LIN {X 0,Y 312.688,Z 247.371,A -85,B 0,C 180,E1 -15958.713,E2 -15958.713} C_VEL
LIN {X 0,Y 312.385,Z 243.779,A -85,B 0,C 180,E1 -15959.666,E2 -15959.666} C_VEL
LIN {X 0,Y 310.267,Z 233.599,A -85,B 0,C 180,E1 -15962.611,E2 -15962.611} C_VEL
LIN {X 0,Y 307.607,Z 223.567,A -85,B 0,C 180,E1 -15965.799,E2 -15965.799} C_VEL
LIN {X 0,Y 305.424,Z 216.441,A -85,B 0,C 180,E1 -15968.279,E2 -15968.279} C_VEL
LIN {X 0,Y 305.436,Z 216.435,A -85,B 0,C 180,E1 -15972.581,E2 -15972.581} C_VEL
LIN {X 0,Y 305.421,Z 216.44,A -85,B 0,C 180,E1 -15976.344,E2 -15976.344} C_VEL
LIN {X 0,Y 305.409,Z 216.437,A -85,B 0,C 180,E1 -15979.884,E2 -15979.884} C_VEL
LIN {X 0,Y 305.462,Z 216.436,A -85,B 0,C 180,E1 -15983.636,E2 -15983.636} C_VEL
LIN {X 0,Y 305.464,Z 216.436,A -85,B 0,C 180,E1 -15986.483,E2 -15986.483} C_VEL
LIN {X 0,Y 305.433,Z 216.439,A -85,B 0,C 180,E1 -15989.587,E2 -15989.587} C_VEL
LIN {X 0,Y 305.466,Z 216.432,A -85,B 0,C 180,E1 -15992.603,E2 -15992.603} C_VEL
LIN {X 0,Y 305.486,Z 216.432,A -85,B 0,C 180,E1 -15995.537,E2 -15995.537} C_VEL
LIN {X 0,Y 305.5,Z 216.426,A -85,B 0,C 180,E1 -15999.814,E2 -15999.814} C_VEL
LIN {X 0,Y 305.546,Z 216.418,A -85,B 0,C 180,E1 -16002.601,E2 -16002.601} C_VEL
LIN {X 0,Y 305.626,Z 216.409,A -85,B 0,C 180,E1 -16005.348,E2 -16005.348} C_VEL
LIN {X 0,Y 305.635,Z 216.412,A -85,B 0,C 180,E1 -16009.4,E2 -16009.4} C_VEL
LIN {X 0,Y 305.797,Z 216.394,A -85,B 0,C 180,E1 -16012.074,E2 -16012.074} C_VEL
LIN {X 0,Y 305.685,Z 216.407,A -85,B 0,C 180,E1 -16014.723,E2 -16014.723} C_VEL
LIN {X 0,Y 305.955,Z 216.371,A -85,B 0,C 180,E1 -16018.684,E2 -16018.684} C_VEL
LIN {X 0,Y 305.955,Z 216.375,A -85,B 0,C 180,E1 -16021.316,E2 -16021.316} C_VEL
LIN {X 0,Y 305.676,Z 216.41,A -85,B 0,C 180,E1 -16025.277,E2 -16025.277} C_VEL
LIN {X 0,Y 305.768,Z 216.397,A -85,B 0,C 180,E1 -16027.927,E2 -16027.927} C_VEL
LIN {X 0,Y 305.773,Z 216.514,A -85,B 0,C 180,E1 -16028.46,E2 -16028.46} C_VEL
LIN {X 0,Y 306.843,Z 219.417,A -85,B 0,C 180,E1 -16028.732,E2 -16028.732} C_VEL
LIN {X 0,Y 308.362,Z 221.654,A -85,B 0,C 180,E1 -16029.043,E2 -16029.043} C_VEL
LIN {X 0,Y 315.915,Z 234.684,A -85,B 0,C 180,E1 -16030.554,E2 -16030.554} C_VEL
LIN {X 0,Y 322.045,Z 246.925,A -85,B 0,C 180,E1 -16031.739,E2 -16031.739} C_VEL
LIN {X 0,Y 323.047,Z 249.102,A -85,B 0,C 180,E1 -16031.928,E2 -16031.928} C_VEL
LIN {X 0,Y 319.984,Z 321.185,A -85,B 0,C 180,E1 -16033.904,E2 -16033.904} C_VEL
LIN {X 0,Y 319.265,Z 334.155,A -85,B 0,C 180,E1 -16034.524,E2 -16034.524} C_VEL
LIN {X 0,Y 318.134,Z 346.76,A -85,B 0,C 180,E1 -16035.373,E2 -16035.373} C_VEL
LIN {X 0,Y 316.667,Z 358.574,A -85,B 0,C 180,E1 -16036.437,E2 -16036.437} C_VEL
LIN {X 0,Y 315.006,Z 370.51,A -85,B 0,C 180,E1 -16037.832,E2 -16037.832} C_VEL
LIN {X 0,Y 313.265,Z 380.5,A -85,B 0,C 180,E1 -16039.301,E2 -16039.301} C_VEL
LIN {X 0,Y 311.413,Z 390.569,A -85,B 0,C 180,E1 -16041.167,E2 -16041.167} C_VEL
LIN {X 0,Y 309.756,Z 398.606,A -85,B 0,C 180,E1 -16043.04,E2 -16043.04} C_VEL
LIN {X 0,Y 308.28,Z 405.247,A -85,B 0,C 180,E1 -16044.985,E2 -16044.985} C_VEL
LIN {X 0,Y 306.948,Z 411.266,A -85,B 0,C 180,E1 -16047.253,E2 -16047.253} C_VEL
LIN {X 0,Y 305.986,Z 415.201,A -85,B 0,C 180,E1 -16049.215,E2 -16049.215} C_VEL
LIN {X 0,Y 305.093,Z 418.533,A -85,B 0,C 180,E1 -16051.536,E2 -16051.536} C_VEL
LIN {X 0,Y 304.455,Z 420.465,A -85,B 0,C 180,E1 -16053.797,E2 -16053.797} C_VEL
LIN {X 0,Y 304.084,Z 421.192,A -85,B 0,C 180,E1 -16056.01,E2 -16056.01} C_VEL
LIN {X 0,Y 303.898,Z 420.598,A -85,B 0,C 180,E1 -16058.639,E2 -16058.639} C_VEL
LIN {X 0,Y 303.963,Z 419.321,A -85,B 0,C 180,E1 -16060.346,E2 -16060.346} C_VEL
LIN {X 0,Y 304.211,Z 416.972,A -85,B 0,C 180,E1 -16062.331,E2 -16062.331} C_VEL
LIN {X 0,Y 304.581,Z 413.591,A -85,B 0,C 180,E1 -16064.332,E2 -16064.332} C_VEL
LIN {X 0,Y 305.07,Z 409.227,A -85,B 0,C 180,E1 -16066.282,E2 -16066.282} C_VEL
LIN {X 0,Y 305.647,Z 403.845,A -85,B 0,C 180,E1 -16068.178,E2 -16068.178} C_VEL
LIN {X 0,Y 306.511,Z 396.159,A -85,B 0,C 180,E1 -16070.333,E2 -16070.333} C_VEL
LIN {X 0,Y 307.543,Z 387.805,A -85,B 0,C 180,E1 -16072.185,E2 -16072.185} C_VEL
LIN {X 0,Y 308.695,Z 377.652,A -85,B 0,C 180,E1 -16074.002,E2 -16074.002} C_VEL
LIN {X 0,Y 309.71,Z 367.705,A -85,B 0,C 180,E1 -16075.438,E2 -16075.438} C_VEL
LIN {X 0,Y 310.869,Z 356.07,A -85,B 0,C 180,E1 -16076.77,E2 -16076.77} C_VEL
LIN {X 0,Y 311.902,Z 343.287,A -85,B 0,C 180,E1 -16077.911,E2 -16077.911} C_VEL
LIN {X 0,Y 312.629,Z 329.893,A -85,B 0,C 180,E1 -16078.784,E2 -16078.784} C_VEL
LIN {X 0,Y 313.199,Z 316.6,A -85,B 0,C 180,E1 -16079.374,E2 -16079.374} C_VEL
LIN {X 0,Y 315.113,Z 241.687,A -85,B 0,C 180,E1 -16081.346,E2 -16081.346} C_VEL
LIN {X 0,Y 305.539,Z 216.426,A -85,B 0,C 180,E1 -16082.7,E2 -16082.7} C_VEL
LIN {X 0,Y 305.505,Z 216.429,A -85,B 0,C 180,E1 -16085.539,E2 -16085.539} C_VEL
LIN {X 0,Y 305.497,Z 216.429,A -85,B 0,C 180,E1 -16089.814,E2 -16089.814} C_VEL
LIN {X 0,Y 305.545,Z 216.425,A -85,B 0,C 180,E1 -16092.602,E2 -16092.602} C_VEL
LIN {X 0,Y 305.627,Z 216.414,A -85,B 0,C 180,E1 -16095.348,E2 -16095.348} C_VEL
LIN {X 0,Y 305.625,Z 216.413,A -85,B 0,C 180,E1 -16099.4,E2 -16099.4} C_VEL
LIN {X 0,Y 305.75,Z 216.398,A -85,B 0,C 180,E1 -16102.073,E2 -16102.073} C_VEL
LIN {X 0,Y 305.672,Z 216.411,A -85,B 0,C 180,E1 -16104.724,E2 -16104.724} C_VEL
LIN {X 0,Y 305.953,Z 216.375,A -85,B 0,C 180,E1 -16108.684,E2 -16108.684} C_VEL
LIN {X 0,Y 305.953,Z 216.371,A -85,B 0,C 180,E1 -16111.317,E2 -16111.317} C_VEL
LIN {X 0,Y 305.669,Z 216.407,A -85,B 0,C 180,E1 -16115.277,E2 -16115.277} C_VEL
LIN {X 0,Y 305.765,Z 216.397,A -85,B 0,C 180,E1 -16117.927,E2 -16117.927} C_VEL
LIN {X 0,Y 305.605,Z 216.417,A -85,B 0,C 180,E1 -16121.945,E2 -16121.945} C_VEL
LIN {X 0,Y 305.64,Z 216.41,A -85,B 0,C 180,E1 -16125.035,E2 -16125.035} C_VEL
LIN {X 0,Y 305.581,Z 216.417,A -85,B 0,C 180,E1 -16128.783,E2 -16128.783} C_VEL
LIN {X 0,Y 305.488,Z 216.428,A -85,B 0,C 180,E1 -16133.04,E2 -16133.04} C_VEL
LIN {X 0,Y 305.477,Z 216.433,A -85,B 0,C 180,E1 -16136.2,E2 -16136.2} C_VEL
LIN {X 0,Y 305.46,Z 216.433,A -85,B 0,C 180,E1 -16139.038,E2 -16139.038} C_VEL
LIN {X 0,Y 305.438,Z 216.438,A -85,B 0,C 180,E1 -16141.953,E2 -16141.953} C_VEL
LIN {X 0,Y 305.464,Z 216.432,A -85,B 0,C 180,E1 -16145.114,E2 -16145.114} C_VEL
LIN {X 0,Y 305.428,Z 216.433,A -85,B 0,C 180,E1 -16148.524,E2 -16148.524} C_VEL
LIN {X 0,Y 305.429,Z 216.438,A -85,B 0,C 180,E1 -16151.859,E2 -16151.859} C_VEL
LIN {X 0,Y 305.401,Z 216.445,A -85,B 0,C 180,E1 -16155.511,E2 -16155.511} C_VEL
LIN {X 0,Y 305.414,Z 216.439,A -85,B 0,C 180,E1 -16158.139,E2 -16158.139} C_VEL
LIN {X 0,Y 305.462,Z 216.434,A -85,B 0,C 180,E1 -16161.595,E2 -16161.595} C_VEL
LIN {X 0,Y 305.464,Z 216.434,A -85,B 0,C 180,E1 -16164.887,E2 -16164.887} C_VEL
LIN {X 0,Y 305.434,Z 216.433,A -85,B 0,C 180,E1 -16166.96,E2 -16166.96} C_VEL
LIN {X 0,Y 304.738,Z 216.524,A -85,B 0,C 180,E1 -16168.061,E2 -16168.061} C_VEL
LIN {X 0,Y 301.878,Z 216.879,A -85,B 0,C 180,E1 -16169.854,E2 -16169.854} C_VEL
LIN {X 0,Y 299.48,Z 217.18,A -85,B 0,C 180,E1 -16171.309,E2 -16171.309} C_VEL
LIN {X 0,Y 298.464,Z 217.305,A -85,B 0,C 180,E1 -16172.435,E2 -16172.435} C_VEL
LIN {X 0,Y 298.387,Z 217.311,A -85,B 0,C 180,E1 -16172.816,E2 -16172.816} C_VEL
LIN {X 0,Y 298.423,Z 217.309,A -85,B 0,C 180,E1 -16176.399,E2 -16176.399} C_VEL
LIN {X 0,Y 298.509,Z 217.303,A -85,B 0,C 180,E1 -16180.755,E2 -16180.755} C_VEL
LIN {X 0,Y 298.589,Z 217.29,A -85,B 0,C 180,E1 -16184.995,E2 -16184.995} C_VEL
LIN {X 0,Y 298.586,Z 217.285,A -85,B 0,C 180,E1 -16189.146,E2 -16189.146} C_VEL
LIN {X 0,Y 298.701,Z 217.271,A -85,B 0,C 180,E1 -16191.884,E2 -16191.884} C_VEL
LIN {X 0,Y 298.637,Z 217.286,A -85,B 0,C 180,E1 -16194.599,E2 -16194.599} C_VEL
LIN {X 0,Y 298.91,Z 217.252,A -85,B 0,C 180,E1 -16198.653,E2 -16198.653} C_VEL
LIN {X 0,Y 298.915,Z 217.248,A -85,B 0,C 180,E1 -16201.347,E2 -16201.347} C_VEL
LIN {X 0,Y 298.738,Z 217.268,A -85,B 0,C 180,E1 -16206.755,E2 -16206.755} C_VEL
LIN {X 0,Y 298.633,Z 217.281,A -85,B 0,C 180,E1 -16209.482,E2 -16209.482} C_VEL
LIN {X 0,Y 298.527,Z 217.298,A -85,B 0,C 180,E1 -16213.617,E2 -16213.617} C_VEL
LIN {X 0,Y 298.5,Z 217.304,A -85,B 0,C 180,E1 -16217.823,E2 -16217.823} C_VEL
LIN {X 0,Y 298.428,Z 217.307,A -85,B 0,C 180,E1 -16220.686,E2 -16220.686} C_VEL
LIN {X 0,Y 298.424,Z 217.31,A -85,B 0,C 180,E1 -16225.082,E2 -16225.082} C_VEL
LIN {X 0,Y 298.404,Z 217.314,A -85,B 0,C 180,E1 -16229.375,E2 -16229.375} C_VEL
LIN {X 0,Y 298.395,Z 217.313,A -85,B 0,C 180,E1 -16232.8,E2 -16232.8} C_VEL
LIN {X 0,Y 298.43,Z 217.309,A -85,B 0,C 180,E1 -16236.803,E2 -16236.803} C_VEL
LIN {X 0,Y 298.376,Z 217.321,A -85,B 0,C 180,E1 -16239.492,E2 -16239.492} C_VEL
LIN {X 0,Y 298.372,Z 217.319,A -85,B 0,C 180,E1 -16243.097,E2 -16243.097} C_VEL
LIN {X 0,Y 298.373,Z 217.318,A -85,B 0,C 180,E1 -16246.915,E2 -16246.915} C_VEL
LIN {X 0,Y 298.387,Z 217.318,A -85,B 0,C 180,E1 -16251.011,E2 -16251.011} C_VEL
LIN {X 0,Y 298.409,Z 217.312,A -85,B 0,C 180,E1 -16253.928,E2 -16253.928} C_VEL
LIN {X 0,Y 298.47,Z 217.477,A -85,B 0,C 180,E1 -16255.589,E2 -16255.589} C_VEL
LIN {X 0,Y 301.208,Z 230.094,A -85,B 0,C 180,E1 -16259.114,E2 -16259.114} C_VEL
LIN {X 0,Y 303.252,Z 240.673,A -85,B 0,C 180,E1 -16261.947,E2 -16261.947} C_VEL
LIN {X 0,Y 301.833,Z 252.558,A -85,B 0,C 180,E1 -16264.843,E2 -16264.843} C_VEL
LIN {X 0,Y 307.37,Z 301.3,A -85,B 0,C 180,E1 -16266.603,E2 -16266.603} C_VEL
LIN {X 0,Y 305.725,Z 362.778,A -85,B 0,C 180,E1 -16268.286,E2 -16268.286} C_VEL
LIN {X 0,Y 304.805,Z 376.523,A -85,B 0,C 180,E1 -16268.927,E2 -16268.927} C_VEL
LIN {X 0,Y 303.869,Z 387.983,A -85,B 0,C 180,E1 -16269.7,E2 -16269.7} C_VEL
LIN {X 0,Y 302.703,Z 399.031,A -85,B 0,C 180,E1 -16270.679,E2 -16270.679} C_VEL
LIN {X 0,Y 301.341,Z 410.628,A -85,B 0,C 180,E1 -16271.999,E2 -16271.999} C_VEL
LIN {X 0,Y 300.091,Z 421.14,A -85,B 0,C 180,E1 -16273.503,E2 -16273.503} C_VEL
LIN {X 0,Y 299.107,Z 429.755,A -85,B 0,C 180,E1 -16275.021,E2 -16275.021} C_VEL
LIN {X 0,Y 298.111,Z 439.072,A -85,B 0,C 180,E1 -16277.058,E2 -16277.058} C_VEL
LIN {X 0,Y 297.307,Z 446.538,A -85,B 0,C 180,E1 -16279.099,E2 -16279.099} C_VEL
LIN {X 0,Y 296.966,Z 452.512,A -85,B 0,C 180,E1 -16281.151,E2 -16281.151} C_VEL
LIN {X 0,Y 296.848,Z 457.164,A -85,B 0,C 180,E1 -16283.201,E2 -16283.201} C_VEL
LIN {X 0,Y 296.877,Z 459.588,A -85,B 0,C 180,E1 -16284.566,E2 -16284.566} C_VEL
LIN {X 0,Y 296.844,Z 461.54,A -85,B 0,C 180,E1 -16285.927,E2 -16285.927} C_VEL
LIN {X 0,Y 296.928,Z 463.054,A -85,B 0,C 180,E1 -16287.286,E2 -16287.286} C_VEL
LIN {X 0,Y 297.085,Z 464.085,A -85,B 0,C 180,E1 -16288.644,E2 -16288.644} C_VEL
LIN {X 0,Y 297.089,Z 464.68,A -85,B 0,C 180,E1 -16290,E2 -16290} C_VEL
LIN {X 0,Y 297.049,Z 464.857,A -85,B 0,C 180,E1 -16291.355,E2 -16291.355} C_VEL
LIN {X 0,Y 296.81,Z 464.596,A -85,B 0,C 180,E1 -16292.714,E2 -16292.714} C_VEL
LIN {X 0,Y 296.759,Z 463.895,A -85,B 0,C 180,E1 -16294.074,E2 -16294.074} C_VEL
LIN {X 0,Y 296.649,Z 462.52,A -85,B 0,C 180,E1 -16295.71,E2 -16295.71} C_VEL
LIN {X 0,Y 296.84,Z 459.301,A -85,B 0,C 180,E1 -16298.167,E2 -16298.167} C_VEL
LIN {X 0,Y 297.197,Z 455.495,A -85,B 0,C 180,E1 -16300.215,E2 -16300.215} C_VEL
LIN {X 0,Y 297.889,Z 450.586,A -85,B 0,C 180,E1 -16302.259,E2 -16302.259} C_VEL
LIN {X 0,Y 299.293,Z 443.267,A -85,B 0,C 180,E1 -16304.621,E2 -16304.621} C_VEL
LIN {X 0,Y 300.685,Z 435.56,A -85,B 0,C 180,E1 -16306.602,E2 -16306.602} C_VEL
LIN {X 0,Y 302.319,Z 427.464,A -85,B 0,C 180,E1 -16308.29,E2 -16308.29} C_VEL
LIN {X 0,Y 304.475,Z 416.739,A -85,B 0,C 180,E1 -16310.081,E2 -16310.081} C_VEL
LIN {X 0,Y 306.557,Z 405.968,A -85,B 0,C 180,E1 -16311.519,E2 -16311.519} C_VEL
LIN {X 0,Y 308.314,Z 395.683,A -85,B 0,C 180,E1 -16312.623,E2 -16312.623} C_VEL
LIN {X 0,Y 310.192,Z 383.601,A -85,B 0,C 180,E1 -16313.624,E2 -16313.624} C_VEL
LIN {X 0,Y 311.711,Z 371.311,A -85,B 0,C 180,E1 -16314.386,E2 -16314.386} C_VEL
LIN {X 0,Y 312.826,Z 358.25,A -85,B 0,C 180,E1 -16314.957,E2 -16314.957} C_VEL
LIN {X 0,Y 315.076,Z 301.694,A -85,B 0,C 180,E1 -16316.543,E2 -16316.543} C_VEL
LIN {X 0,Y 312.642,Z 279.918,A -85,B 0,C 180,E1 -16317.569,E2 -16317.569} C_VEL
LIN {X 0,Y 309.361,Z 260.607,A -85,B 0,C 180,E1 -16318.667,E2 -16318.667} C_VEL
LIN {X 0,Y 306.799,Z 249.329,A -85,B 0,C 180,E1 -16319.425,E2 -16319.425} C_VEL
LIN {X 0,Y 305.838,Z 246.569,A -85,B 0,C 180,E1 -16319.712,E2 -16319.712} C_VEL
LIN {X 0,Y 303.74,Z 236.256,A -85,B 0,C 180,E1 -16322.775,E2 -16322.775} C_VEL
LIN {X 0,Y 301.472,Z 227.417,A -85,B 0,C 180,E1 -16325.648,E2 -16325.648} C_VEL
LIN {X 0,Y 298.972,Z 219.432,A -85,B 0,C 180,E1 -16328.521,E2 -16328.521} C_VEL
LIN {X 0,Y 298.356,Z 217.318,A -85,B 0,C 180,E1 -16329.337,E2 -16329.337} C_VEL
LIN {X 0,Y 298.371,Z 217.314,A -85,B 0,C 180,E1 -16333.097,E2 -16333.097} C_VEL
LIN {X 0,Y 298.371,Z 217.314,A -85,B 0,C 180,E1 -16336.915,E2 -16336.915} C_VEL
LIN {X 0,Y 298.384,Z 217.318,A -85,B 0,C 180,E1 -16341.011,E2 -16341.011} C_VEL
LIN {X 0,Y 298.405,Z 217.316,A -85,B 0,C 180,E1 -16343.928,E2 -16343.928} C_VEL
LIN {X 0,Y 298.392,Z 217.312,A -85,B 0,C 180,E1 -16347.199,E2 -16347.199} C_VEL
LIN {X 0,Y 298.407,Z 217.308,A -85,B 0,C 180,E1 -16350.623,E2 -16350.623} C_VEL
LIN {X 0,Y 298.447,Z 217.309,A -85,B 0,C 180,E1 -16354.92,E2 -16354.92} C_VEL
LIN {X 0,Y 298.432,Z 217.306,A -85,B 0,C 180,E1 -16359.314,E2 -16359.314} C_VEL
LIN {X 0,Y 298.507,Z 217.296,A -85,B 0,C 180,E1 -16362.177,E2 -16362.177} C_VEL
LIN {X 0,Y 298.585,Z 217.287,A -85,B 0,C 180,E1 -16364.994,E2 -16364.994} C_VEL
LIN {X 0,Y 298.591,Z 217.288,A -85,B 0,C 180,E1 -16369.146,E2 -16369.146} C_VEL
LIN {X 0,Y 298.741,Z 217.271,A -85,B 0,C 180,E1 -16371.885,E2 -16371.885} C_VEL
LIN {X 0,Y 298.656,Z 217.283,A -85,B 0,C 180,E1 -16374.599,E2 -16374.599} C_VEL
LIN {X 0,Y 298.922,Z 217.247,A -85,B 0,C 180,E1 -16378.653,E2 -16378.653} C_VEL
LIN {X 0,Y 298.922,Z 217.251,A -85,B 0,C 180,E1 -16381.347,E2 -16381.347} C_VEL
LIN {X 0,Y 298.72,Z 217.274,A -85,B 0,C 180,E1 -16386.515,E2 -16386.515} C_VEL
LIN {X 0,Y 298.735,Z 217.275,A -85,B 0,C 180,E1 -16387.349,E2 -16387.349} C_VEL
LIN {X 0,Y 299.806,Z 220.259,A -85,B 0,C 180,E1 -16387.662,E2 -16387.662} C_VEL
LIN {X 0,Y 301.416,Z 222.354,A -85,B 0,C 180,E1 -16388,E2 -16388} C_VEL
LIN {X 0,Y 310.025,Z 237.229,A -85,B 0,C 180,E1 -16389.843,E2 -16389.843} C_VEL
LIN {X 0,Y 316.356,Z 249.735,A -85,B 0,C 180,E1 -16391.123,E2 -16391.123} C_VEL
LIN {X 0,Y 317.022,Z 251.251,A -85,B 0,C 180,E1 -16391.261,E2 -16391.261} C_VEL
LIN {X 0,Y 313.904,Z 322.243,A -85,B 0,C 180,E1 -16393.267,E2 -16393.267} C_VEL
LIN {X 0,Y 313.163,Z 334.721,A -85,B 0,C 180,E1 -16393.878,E2 -16393.878} C_VEL
LIN {X 0,Y 311.958,Z 347.565,A -85,B 0,C 180,E1 -16394.761,E2 -16394.761} C_VEL
LIN {X 0,Y 310.296,Z 360.242,A -85,B 0,C 180,E1 -16395.939,E2 -16395.939} C_VEL
LIN {X 0,Y 308.695,Z 370.876,A -85,B 0,C 180,E1 -16397.216,E2 -16397.216} C_VEL
LIN {X 0,Y 306.904,Z 380.791,A -85,B 0,C 180,E1 -16398.699,E2 -16398.699} C_VEL
LIN {X 0,Y 304.949,Z 390.754,A -85,B 0,C 180,E1 -16400.577,E2 -16400.577} C_VEL
LIN {X 0,Y 303.053,Z 399.391,A -85,B 0,C 180,E1 -16402.624,E2 -16402.624} C_VEL
LIN {X 0,Y 301.351,Z 406.616,A -85,B 0,C 180,E1 -16404.821,E2 -16404.821} C_VEL
LIN {X 0,Y 299.976,Z 412.353,A -85,B 0,C 180,E1 -16407.092,E2 -16407.092} C_VEL
LIN {X 0,Y 298.761,Z 416.929,A -85,B 0,C 180,E1 -16409.604,E2 -16409.604} C_VEL
LIN {X 0,Y 297.919,Z 419.716,A -85,B 0,C 180,E1 -16411.87,E2 -16411.87} C_VEL
LIN {X 0,Y 297.231,Z 421.484,A -85,B 0,C 180,E1 -16414.574,E2 -16414.574} C_VEL
LIN {X 0,Y 296.957,Z 421.761,A -85,B 0,C 180,E1 -16416.422,E2 -16416.422} C_VEL
LIN {X 0,Y 296.822,Z 421.096,A -85,B 0,C 180,E1 -16418.615,E2 -16418.615} C_VEL
LIN {X 0,Y 296.907,Z 419.404,A -85,B 0,C 180,E1 -16420.759,E2 -16420.759} C_VEL
LIN {X 0,Y 297.307,Z 416.024,A -85,B 0,C 180,E1 -16423.277,E2 -16423.277} C_VEL
LIN {X 0,Y 297.669,Z 412.624,A -85,B 0,C 180,E1 -16425.097,E2 -16425.097} C_VEL
LIN {X 0,Y 298.273,Z 406.939,A -85,B 0,C 180,E1 -16427.411,E2 -16427.411} C_VEL
LIN {X 0,Y 298.956,Z 401.062,A -85,B 0,C 180,E1 -16429.293,E2 -16429.293} C_VEL
LIN {X 0,Y 300.017,Z 392.542,A -85,B 0,C 180,E1 -16431.473,E2 -16431.473} C_VEL
LIN {X 0,Y 301.055,Z 383.725,A -85,B 0,C 180,E1 -16433.272,E2 -16433.272} C_VEL
LIN {X 0,Y 302.261,Z 373.726,A -85,B 0,C 180,E1 -16434.926,E2 -16434.926} C_VEL
LIN {X 0,Y 303.359,Z 362.693,A -85,B 0,C 180,E1 -16436.391,E2 -16436.391} C_VEL
LIN {X 0,Y 304.496,Z 350.668,A -85,B 0,C 180,E1 -16437.644,E2 -16437.644} C_VEL
LIN {X 0,Y 305.392,Z 338.484,A -85,B 0,C 180,E1 -16438.623,E2 -16438.623} C_VEL
LIN {X 0,Y 305.993,Z 324.851,A -85,B 0,C 180,E1 -16439.411,E2 -16439.411} C_VEL
LIN {X 0,Y 306.502,Z 311.68,A -85,B 0,C 180,E1 -16439.896,E2 -16439.896} C_VEL
LIN {X 0,Y 308.451,Z 243.989,A -85,B 0,C 180,E1 -16441.693,E2 -16441.693} C_VEL
LIN {X 0,Y 302.906,Z 228.819,A -85,B 0,C 180,E1 -16442.493,E2 -16442.493} C_VEL
LIN {X 0,Y 298.655,Z 218.077,A -85,B 0,C 180,E1 -16443.103,E2 -16443.103} C_VEL
LIN {X 0,Y 298.53,Z 217.3,A -85,B 0,C 180,E1 -16443.175,E2 -16443.175} C_VEL
LIN {X 0,Y 298.431,Z 217.312,A -85,B 0,C 180,E1 -16446.7,E2 -16446.7} C_VEL
LIN {X 0,Y 298.506,Z 217.303,A -85,B 0,C 180,E1 -16450.755,E2 -16450.755} C_VEL
LIN {X 0,Y 298.586,Z 217.293,A -85,B 0,C 180,E1 -16454.995,E2 -16454.995} C_VEL
LIN {X 0,Y 298.584,Z 217.292,A -85,B 0,C 180,E1 -16459.147,E2 -16459.147} C_VEL
LIN {X 0,Y 298.701,Z 217.275,A -85,B 0,C 180,E1 -16461.885,E2 -16461.885} C_VEL
LIN {X 0,Y 298.64,Z 217.287,A -85,B 0,C 180,E1 -16464.599,E2 -16464.599} C_VEL
LIN {X 0,Y 298.92,Z 217.252,A -85,B 0,C 180,E1 -16468.653,E2 -16468.653} C_VEL
LIN {X 0,Y 298.919,Z 217.247,A -85,B 0,C 180,E1 -16471.348,E2 -16471.348} C_VEL
LIN {X 0,Y 298.747,Z 217.271,A -85,B 0,C 180,E1 -16476.755,E2 -16476.755} C_VEL
LIN {X 0,Y 298.632,Z 217.283,A -85,B 0,C 180,E1 -16479.482,E2 -16479.482} C_VEL
LIN {X 0,Y 298.554,Z 217.294,A -85,B 0,C 180,E1 -16483.616,E2 -16483.616} C_VEL
LIN {X 0,Y 298.55,Z 217.296,A -85,B 0,C 180,E1 -16486.409,E2 -16486.409} C_VEL
LIN {X 0,Y 298.499,Z 217.301,A -85,B 0,C 180,E1 -16489.648,E2 -16489.648} C_VEL
LIN {X 0,Y 298.426,Z 217.309,A -85,B 0,C 180,E1 -16493.601,E2 -16493.601} C_VEL
LIN {X 0,Y 298.415,Z 217.311,A -85,B 0,C 180,E1 -16496.582,E2 -16496.582} C_VEL
LIN {X 0,Y 298.399,Z 217.316,A -85,B 0,C 180,E1 -16499.644,E2 -16499.644} C_VEL
LIN {X 0,Y 298.394,Z 217.312,A -85,B 0,C 180,E1 -16502.801,E2 -16502.801} C_VEL
LIN {X 0,Y 298.43,Z 217.305,A -85,B 0,C 180,E1 -16506.803,E2 -16506.803} C_VEL
LIN {X 0,Y 298.383,Z 217.313,A -85,B 0,C 180,E1 -16511.087,E2 -16511.087} C_VEL
LIN {X 0,Y 298.401,Z 217.313,A -85,B 0,C 180,E1 -16513.104,E2 -16513.104} C_VEL
LIN {X 0,Y 298.373,Z 217.317,A -85,B 0,C 180,E1 -16516.915,E2 -16516.915} C_VEL
LIN {X 0,Y 298.386,Z 217.316,A -85,B 0,C 180,E1 -16521.011,E2 -16521.011} C_VEL
LIN {X 0,Y 298.418,Z 217.309,A -85,B 0,C 180,E1 -16523.93,E2 -16523.93} C_VEL
LIN {X 0,Y 298.395,Z 217.318,A -85,B 0,C 180,E1 -16527.2,E2 -16527.2} C_VEL
LIN {X 0,Y 298.405,Z 217.313,A -85,B 0,C 180,E1 -16530.625,E2 -16530.625} C_VEL
LIN {X 0,Y 298.387,Z 217.311,A -85,B 0,C 180,E1 -16532.816,E2 -16532.816} C_VEL
LIN {X 0,Y 297.737,Z 217.396,A -85,B 0,C 180,E1 -16533.943,E2 -16533.943} C_VEL
LIN {X 0,Y 294.9,Z 217.759,A -85,B 0,C 180,E1 -16535.779,E2 -16535.779} C_VEL
LIN {X 0,Y 292.484,Z 218.062,A -85,B 0,C 180,E1 -16537.269,E2 -16537.269} C_VEL
LIN {X 0,Y 291.446,Z 218.186,A -85,B 0,C 180,E1 -16538.423,E2 -16538.423} C_VEL
LIN {X 0,Y 291.361,Z 218.193,A -85,B 0,C 180,E1 -16538.814,E2 -16538.814} C_VEL
LIN {X 0,Y 291.444,Z 218.178,A -85,B 0,C 180,E1 -16541.731,E2 -16541.731} C_VEL
LIN {X 0,Y 291.519,Z 218.168,A -85,B 0,C 180,E1 -16546.05,E2 -16546.05} C_VEL
LIN {X 0,Y 291.571,Z 218.159,A -85,B 0,C 180,E1 -16550.286,E2 -16550.286} C_VEL
LIN {X 0,Y 291.691,Z 218.146,A -85,B 0,C 180,E1 -16553.081,E2 -16553.081} C_VEL
LIN {X 0,Y 291.779,Z 218.137,A -85,B 0,C 180,E1 -16557.239,E2 -16557.239} C_VEL
LIN {X 0,Y 291.863,Z 218.129,A -85,B 0,C 180,E1 -16560,E2 -16560} C_VEL
LIN {X 0,Y 291.765,Z 218.139,A -85,B 0,C 180,E1 -16562.761,E2 -16562.761} C_VEL
LIN {X 0,Y 291.69,Z 218.144,A -85,B 0,C 180,E1 -16566.919,E2 -16566.919} C_VEL
LIN {X 0,Y 291.575,Z 218.161,A -85,B 0,C 180,E1 -16569.714,E2 -16569.714} C_VEL
LIN {X 0,Y 291.485,Z 218.178,A -85,B 0,C 180,E1 -16573.952,E2 -16573.952} C_VEL
LIN {X 0,Y 291.437,Z 218.181,A -85,B 0,C 180,E1 -16578.27,E2 -16578.27} C_VEL
LIN {X 0,Y 291.352,Z 218.188,A -85,B 0,C 180,E1 -16581.213,E2 -16581.213} C_VEL
LIN {X 0,Y 291.336,Z 218.194,A -85,B 0,C 180,E1 -16584.211,E2 -16584.211} C_VEL
LIN {X 0,Y 291.353,Z 218.192,A -85,B 0,C 180,E1 -16587.279,E2 -16587.279} C_VEL
LIN {X 0,Y 291.321,Z 218.193,A -85,B 0,C 180,E1 -16590.439,E2 -16590.439} C_VEL
LIN {X 0,Y 291.346,Z 218.195,A -85,B 0,C 180,E1 -16593.698,E2 -16593.698} C_VEL
LIN {X 0,Y 291.362,Z 218.192,A -85,B 0,C 180,E1 -16597.249,E2 -16597.249} C_VEL
LIN {X 0,Y 291.302,Z 218.198,A -85,B 0,C 180,E1 -16600.648,E2 -16600.648} C_VEL
LIN {X 0,Y 291.283,Z 218.2,A -85,B 0,C 180,E1 -16604.403,E2 -16604.403} C_VEL
LIN {X 0,Y 291.297,Z 218.198,A -85,B 0,C 180,E1 -16608.411,E2 -16608.411} C_VEL
LIN {X 0,Y 291.337,Z 218.197,A -85,B 0,C 180,E1 -16611.155,E2 -16611.155} C_VEL
LIN {X 0,Y 291.383,Z 218.189,A -85,B 0,C 180,E1 -16614.629,E2 -16614.629} C_VEL
LIN {X 0,Y 291.414,Z 218.323,A -85,B 0,C 180,E1 -16615.215,E2 -16615.215} C_VEL
LIN {X 0,Y 294.135,Z 230.993,A -85,B 0,C 180,E1 -16618.842,E2 -16618.842} C_VEL
LIN {X 0,Y 296.221,Z 241.276,A -85,B 0,C 180,E1 -16621.672,E2 -16621.672} C_VEL
LIN {X 0,Y 295.423,Z 248.76,A -85,B 0,C 180,E1 -16623.547,E2 -16623.547} C_VEL
LIN {X 0,Y 294.987,Z 252.087,A -85,B 0,C 180,E1 -16624.374,E2 -16624.374} C_VEL
LIN {X 0,Y 300.595,Z 301.672,A -85,B 0,C 180,E1 -16626.218,E2 -16626.218} C_VEL
LIN {X 0,Y 298.911,Z 361.828,A -85,B 0,C 180,E1 -16627.902,E2 -16627.902} C_VEL
LIN {X 0,Y 298.06,Z 374.978,A -85,B 0,C 180,E1 -16628.517,E2 -16628.517} C_VEL
LIN {X 0,Y 296.977,Z 387.769,A -85,B 0,C 180,E1 -16629.389,E2 -16629.389} C_VEL
LIN {X 0,Y 295.57,Z 400.313,A -85,B 0,C 180,E1 -16630.555,E2 -16630.555} C_VEL
LIN {X 0,Y 294.254,Z 411.607,A -85,B 0,C 180,E1 -16631.911,E2 -16631.911} C_VEL
LIN {X 0,Y 293.106,Z 420.782,A -85,B 0,C 180,E1 -16633.277,E2 -16633.277} C_VEL
LIN {X 0,Y 292.143,Z 428.459,A -85,B 0,C 180,E1 -16634.655,E2 -16634.655} C_VEL
LIN {X 0,Y 291.25,Z 436.544,A -85,B 0,C 180,E1 -16636.392,E2 -16636.392} C_VEL
LIN {X 0,Y 290.548,Z 443.221,A -85,B 0,C 180,E1 -16638.135,E2 -16638.135} C_VEL
LIN {X 0,Y 290.021,Z 449.751,A -85,B 0,C 180,E1 -16640.233,E2 -16640.233} C_VEL
LIN {X 0,Y 289.792,Z 454.898,A -85,B 0,C 180,E1 -16642.334,E2 -16642.334} C_VEL
LIN {X 0,Y 289.809,Z 458.841,A -85,B 0,C 180,E1 -16644.433,E2 -16644.433} C_VEL
LIN {X 0,Y 289.776,Z 460.83,A -85,B 0,C 180,E1 -16645.827,E2 -16645.827} C_VEL
LIN {X 0,Y 289.84,Z 462.382,A -85,B 0,C 180,E1 -16647.22,E2 -16647.22} C_VEL
LIN {X 0,Y 290.024,Z 463.475,A -85,B 0,C 180,E1 -16648.611,E2 -16648.611} C_VEL
LIN {X 0,Y 290.032,Z 464.101,A -85,B 0,C 180,E1 -16650,E2 -16650} C_VEL
LIN {X 0,Y 289.966,Z 464.305,A -85,B 0,C 180,E1 -16651.388,E2 -16651.388} C_VEL
LIN {X 0,Y 289.722,Z 464.086,A -85,B 0,C 180,E1 -16652.78,E2 -16652.78} C_VEL
LIN {X 0,Y 289.659,Z 463.431,A -85,B 0,C 180,E1 -16654.174,E2 -16654.174} C_VEL
LIN {X 0,Y 289.602,Z 460.866,A -85,B 0,C 180,E1 -16656.969,E2 -16656.969} C_VEL
LIN {X 0,Y 289.866,Z 457.817,A -85,B 0,C 180,E1 -16659.067,E2 -16659.067} C_VEL
LIN {X 0,Y 290.333,Z 453.726,A -85,B 0,C 180,E1 -16661.166,E2 -16661.166} C_VEL
LIN {X 0,Y 291.534,Z 447.542,A -85,B 0,C 180,E1 -16663.594,E2 -16663.594} C_VEL
LIN {X 0,Y 292.861,Z 440.803,A -85,B 0,C 180,E1 -16665.657,E2 -16665.657} C_VEL
LIN {X 0,Y 294.54,Z 432.463,A -85,B 0,C 180,E1 -16667.711,E2 -16667.711} C_VEL
LIN {X 0,Y 296.366,Z 424.071,A -85,B 0,C 180,E1 -16669.39,E2 -16669.39} C_VEL
LIN {X 0,Y 298.552,Z 413.913,A -85,B 0,C 180,E1 -16671.038,E2 -16671.038} C_VEL
LIN {X 0,Y 300.72,Z 402.553,A -85,B 0,C 180,E1 -16672.5,E2 -16672.5} C_VEL
LIN {X 0,Y 302.955,Z 389.824,A -85,B 0,C 180,E1 -16673.77,E2 -16673.77} C_VEL
LIN {X 0,Y 304.787,Z 377.212,A -85,B 0,C 180,E1 -16674.704,E2 -16674.704} C_VEL
LIN {X 0,Y 306.245,Z 364.261,A -85,B 0,C 180,E1 -16675.395,E2 -16675.395} C_VEL
LIN {X 0,Y 307.144,Z 351.021,A -85,B 0,C 180,E1 -16675.863,E2 -16675.863} C_VEL
LIN {X 0,Y 309.165,Z 302.802,A -85,B 0,C 180,E1 -16677.234,E2 -16677.234} C_VEL
LIN {X 0,Y 306.836,Z 281.371,A -85,B 0,C 180,E1 -16678.284,E2 -16678.284} C_VEL
LIN {X 0,Y 303.474,Z 261.317,A -85,B 0,C 180,E1 -16679.468,E2 -16679.468} C_VEL
LIN {X 0,Y 301.389,Z 252.243,A -85,B 0,C 180,E1 -16680.119,E2 -16680.119} C_VEL
LIN {X 0,Y 298.688,Z 245.762,A -85,B 0,C 180,E1 -16680.832,E2 -16680.832} C_VEL
LIN {X 0,Y 296.523,Z 235.859,A -85,B 0,C 180,E1 -16683.947,E2 -16683.947} C_VEL
LIN {X 0,Y 294.036,Z 226.803,A -85,B 0,C 180,E1 -16687.097,E2 -16687.097} C_VEL
LIN {X 0,Y 291.3,Z 218.197,A -85,B 0,C 180,E1 -16690.484,E2 -16690.484} C_VEL
LIN {X 0,Y 291.282,Z 218.199,A -85,B 0,C 180,E1 -16694.403,E2 -16694.403} C_VEL
LIN {X 0,Y 291.295,Z 218.199,A -85,B 0,C 180,E1 -16698.411,E2 -16698.411} C_VEL
LIN {X 0,Y 291.335,Z 218.196,A -85,B 0,C 180,E1 -16701.155,E2 -16701.155} C_VEL
LIN {X 0,Y 291.355,Z 218.188,A -85,B 0,C 180,E1 -16704.625,E2 -16704.625} C_VEL
LIN {X 0,Y 291.366,Z 218.186,A -85,B 0,C 180,E1 -16707.95,E2 -16707.95} C_VEL
LIN {X 0,Y 291.351,Z 218.189,A -85,B 0,C 180,E1 -16711.155,E2 -16711.155} C_VEL
LIN {X 0,Y 291.374,Z 218.187,A -85,B 0,C 180,E1 -16714.268,E2 -16714.268} C_VEL
LIN {X 0,Y 291.372,Z 218.188,A -85,B 0,C 180,E1 -16717.299,E2 -16717.299} C_VEL
LIN {X 0,Y 291.458,Z 218.177,A -85,B 0,C 180,E1 -16720.27,E2 -16720.27} C_VEL
LIN {X 0,Y 291.514,Z 218.17,A -85,B 0,C 180,E1 -16724.653,E2 -16724.653} C_VEL
LIN {X 0,Y 291.535,Z 218.165,A -85,B 0,C 180,E1 -16728.88,E2 -16728.88} C_VEL
LIN {X 0,Y 291.688,Z 218.148,A -85,B 0,C 180,E1 -16731.688,E2 -16731.688} C_VEL
LIN {X 0,Y 291.626,Z 218.158,A -85,B 0,C 180,E1 -16734.468,E2 -16734.468} C_VEL
LIN {X 0,Y 291.888,Z 218.123,A -85,B 0,C 180,E1 -16738.62,E2 -16738.62} C_VEL
LIN {X 0,Y 291.888,Z 218.127,A -85,B 0,C 180,E1 -16741.38,E2 -16741.38} C_VEL
LIN {X 0,Y 291.662,Z 218.154,A -85,B 0,C 180,E1 -16746.138,E2 -16746.138} C_VEL
LIN {X 0,Y 292.663,Z 220.956,A -85,B 0,C 180,E1 -16746.463,E2 -16746.463} C_VEL
LIN {X 0,Y 294.545,Z 223.309,A -85,B 0,C 180,E1 -16746.893,E2 -16746.893} C_VEL
LIN {X 0,Y 296.569,Z 226.612,A -85,B 0,C 180,E1 -16747.376,E2 -16747.376} C_VEL
LIN {X 0,Y 304.765,Z 240.757,A -85,B 0,C 180,E1 -16749.21,E2 -16749.21} C_VEL
LIN {X 0,Y 311.112,Z 253.364,A -85,B 0,C 180,E1 -16750.555,E2 -16750.555} C_VEL
LIN {X 0,Y 307.937,Z 322.519,A -85,B 0,C 180,E1 -16752.563,E2 -16752.563} C_VEL
LIN {X 0,Y 307.118,Z 335.085,A -85,B 0,C 180,E1 -16753.186,E2 -16753.186} C_VEL
LIN {X 0,Y 305.917,Z 347.401,A -85,B 0,C 180,E1 -16754.043,E2 -16754.043} C_VEL
LIN {X 0,Y 304.45,Z 358.478,A -85,B 0,C 180,E1 -16755.052,E2 -16755.052} C_VEL
LIN {X 0,Y 302.604,Z 370.357,A -85,B 0,C 180,E1 -16756.456,E2 -16756.456} C_VEL
LIN {X 0,Y 300.575,Z 381.035,A -85,B 0,C 180,E1 -16758.048,E2 -16758.048} C_VEL
LIN {X 0,Y 298.728,Z 390.148,A -85,B 0,C 180,E1 -16759.771,E2 -16759.771} C_VEL
LIN {X 0,Y 296.627,Z 399.23,A -85,B 0,C 180,E1 -16761.911,E2 -16761.911} C_VEL
LIN {X 0,Y 294.967,Z 405.835,A -85,B 0,C 180,E1 -16763.894,E2 -16763.894} C_VEL
LIN {X 0,Y 293.378,Z 412.059,A -85,B 0,C 180,E1 -16766.307,E2 -16766.307} C_VEL
LIN {X 0,Y 292.053,Z 416.775,A -85,B 0,C 180,E1 -16768.769,E2 -16768.769} C_VEL
LIN {X 0,Y 291.377,Z 419.055,A -85,B 0,C 180,E1 -16770.432,E2 -16770.432} C_VEL
LIN {X 0,Y 290.747,Z 420.834,A -85,B 0,C 180,E1 -16772.218,E2 -16772.218} C_VEL
LIN {X 0,Y 290.17,Z 422.097,A -85,B 0,C 180,E1 -16774.565,E2 -16774.565} C_VEL
LIN {X 0,Y 289.806,Z 422.115,A -85,B 0,C 180,E1 -16777.32,E2 -16777.32} C_VEL
LIN {X 0,Y 289.732,Z 421.244,A -85,B 0,C 180,E1 -16779.1,E2 -16779.1} C_VEL
LIN {X 0,Y 289.884,Z 419.281,A -85,B 0,C 180,E1 -16781.274,E2 -16781.274} C_VEL
LIN {X 0,Y 290.254,Z 416.311,A -85,B 0,C 180,E1 -16783.415,E2 -16783.415} C_VEL
LIN {X 0,Y 290.785,Z 411.469,A -85,B 0,C 180,E1 -16785.911,E2 -16785.911} C_VEL
LIN {X 0,Y 291.376,Z 406.453,A -85,B 0,C 180,E1 -16787.868,E2 -16787.868} C_VEL
LIN {X 0,Y 292.145,Z 399.825,A -85,B 0,C 180,E1 -16789.934,E2 -16789.934} C_VEL
LIN {X 0,Y 293.303,Z 391.042,A -85,B 0,C 180,E1 -16792.108,E2 -16792.108} C_VEL
LIN {X 0,Y 294.307,Z 382.588,A -85,B 0,C 180,E1 -16793.804,E2 -16793.804} C_VEL
LIN {X 0,Y 295.513,Z 372.439,A -85,B 0,C 180,E1 -16795.454,E2 -16795.454} C_VEL
LIN {X 0,Y 296.563,Z 362.253,A -85,B 0,C 180,E1 -16796.796,E2 -16796.796} C_VEL
LIN {X 0,Y 297.745,Z 349.726,A -85,B 0,C 180,E1 -16798.104,E2 -16798.104} C_VEL
LIN {X 0,Y 298.647,Z 337.246,A -85,B 0,C 180,E1 -16799.084,E2 -16799.084} C_VEL
LIN {X 0,Y 299.273,Z 323.521,A -85,B 0,C 180,E1 -16799.861,E2 -16799.861} C_VEL
LIN {X 0,Y 299.718,Z 310.07,A -85,B 0,C 180,E1 -16800.33,E2 -16800.33} C_VEL
LIN {X 0,Y 301.702,Z 245.201,A -85,B 0,C 180,E1 -16802.091,E2 -16802.091} C_VEL
LIN {X 0,Y 294.399,Z 226.058,A -85,B 0,C 180,E1 -16803.163,E2 -16803.163} C_VEL
LIN {X 0,Y 291.443,Z 218.182,A -85,B 0,C 180,E1 -16803.623,E2 -16803.623} C_VEL
LIN {X 0,Y 291.373,Z 218.191,A -85,B 0,C 180,E1 -16807.299,E2 -16807.299} C_VEL
LIN {X 0,Y 291.439,Z 218.18,A -85,B 0,C 180,E1 -16810.269,E2 -16810.269} C_VEL
LIN {X 0,Y 291.498,Z 218.176,A -85,B 0,C 180,E1 -16814.666,E2 -16814.666} C_VEL
LIN {X 0,Y 291.53,Z 218.173,A -85,B 0,C 180,E1 -16818.881,E2 -16818.881} C_VEL
LIN {X 0,Y 291.654,Z 218.153,A -85,B 0,C 180,E1 -16821.687,E2 -16821.687} C_VEL
LIN {X 0,Y 291.609,Z 218.162,A -85,B 0,C 180,E1 -16824.468,E2 -16824.468} C_VEL
LIN {X 0,Y 291.886,Z 218.128,A -85,B 0,C 180,E1 -16828.621,E2 -16828.621} C_VEL
LIN {X 0,Y 291.886,Z 218.124,A -85,B 0,C 180,E1 -16831.38,E2 -16831.38} C_VEL
LIN {X 0,Y 291.699,Z 218.148,A -85,B 0,C 180,E1 -16836.919,E2 -16836.919} C_VEL
LIN {X 0,Y 291.573,Z 218.163,A -85,B 0,C 180,E1 -16839.714,E2 -16839.714} C_VEL
LIN {X 0,Y 291.524,Z 218.172,A -85,B 0,C 180,E1 -16843.951,E2 -16843.951} C_VEL
LIN {X 0,Y 291.488,Z 218.174,A -85,B 0,C 180,E1 -16846.818,E2 -16846.818} C_VEL
LIN {X 0,Y 291.452,Z 218.18,A -85,B 0,C 180,E1 -16849.875,E2 -16849.875} C_VEL
LIN {X 0,Y 291.368,Z 218.19,A -85,B 0,C 180,E1 -16854.209,E2 -16854.209} C_VEL
LIN {X 0,Y 291.361,Z 218.19,A -85,B 0,C 180,E1 -16857.278,E2 -16857.278} C_VEL
LIN {X 0,Y 291.322,Z 218.194,A -85,B 0,C 180,E1 -16860.439,E2 -16860.439} C_VEL
LIN {X 0,Y 291.345,Z 218.193,A -85,B 0,C 180,E1 -16863.699,E2 -16863.699} C_VEL
LIN {X 0,Y 291.359,Z 218.186,A -85,B 0,C 180,E1 -16867.25,E2 -16867.25} C_VEL
LIN {X 0,Y 291.329,Z 218.189,A -85,B 0,C 180,E1 -16870.644,E2 -16870.644} C_VEL
LIN {X 0,Y 291.292,Z 218.197,A -85,B 0,C 180,E1 -16874.402,E2 -16874.402} C_VEL
LIN {X 0,Y 291.297,Z 218.197,A -85,B 0,C 180,E1 -16878.412,E2 -16878.412} C_VEL
LIN {X 0,Y 291.337,Z 218.195,A -85,B 0,C 180,E1 -16881.156,E2 -16881.156} C_VEL
LIN {X 0,Y 291.362,Z 218.188,A -85,B 0,C 180,E1 -16884.626,E2 -16884.626} C_VEL
LIN {X 0,Y 291.368,Z 218.188,A -85,B 0,C 180,E1 -16887.95,E2 -16887.95} C_VEL
LIN {X 0,Y 291.347,Z 218.194,A -85,B 0,C 180,E1 -16891.155,E2 -16891.155} C_VEL
LIN {X 0,Y 291.361,Z 218.188,A -85,B 0,C 180,E1 -16894.267,E2 -16894.267} C_VEL
LIN {X 0,Y 291.373,Z 218.189,A -85,B 0,C 180,E1 -16897.299,E2 -16897.299} C_VEL
LIN {X 0,Y 291.361,Z 218.193,A -85,B 0,C 180,E1 -16898.814,E2 -16898.814} C_VEL
LIN {X 0,Y 290.705,Z 218.272,A -85,B 0,C 180,E1 -16899.968,E2 -16899.968} C_VEL
LIN {X 0,Y 287.902,Z 218.619,A -85,B 0,C 180,E1 -16901.851,E2 -16901.851} C_VEL
LIN {X 0,Y 285.531,Z 218.917,A -85,B 0,C 180,E1 -16903.379,E2 -16903.379} C_VEL
LIN {X 0,Y 284.52,Z 219.043,A -85,B 0,C 180,E1 -16904.561,E2 -16904.561} C_VEL
LIN {X 0,Y 284.442,Z 219.049,A -85,B 0,C 180,E1 -16904.962,E2 -16904.962} C_VEL
LIN {X 0,Y 284.485,Z 219.043,A -85,B 0,C 180,E1 -16908.601,E2 -16908.601} C_VEL
LIN {X 0,Y 284.611,Z 219.023,A -85,B 0,C 180,E1 -16911.48,E2 -16911.48} C_VEL
LIN {X 0,Y 284.576,Z 219.034,A -85,B 0,C 180,E1 -16914.331,E2 -16914.331} C_VEL
LIN {X 0,Y 284.845,Z 219.004,A -85,B 0,C 180,E1 -16918.586,E2 -16918.586} C_VEL
LIN {X 0,Y 284.848,Z 219,A -85,B 0,C 180,E1 -16921.414,E2 -16921.414} C_VEL
LIN {X 0,Y 284.645,Z 219.021,A -85,B 0,C 180,E1 -16927.091,E2 -16927.091} C_VEL
LIN {X 0,Y 284.52,Z 219.041,A -85,B 0,C 180,E1 -16929.957,E2 -16929.957} C_VEL
LIN {X 0,Y 284.438,Z 219.055,A -85,B 0,C 180,E1 -16934.305,E2 -16934.305} C_VEL
LIN {X 0,Y 284.373,Z 219.059,A -85,B 0,C 180,E1 -16938.741,E2 -16938.741} C_VEL
LIN {X 0,Y 284.305,Z 219.069,A -85,B 0,C 180,E1 -16941.765,E2 -16941.765} C_VEL
LIN {X 0,Y 284.291,Z 219.07,A -85,B 0,C 180,E1 -16944.851,E2 -16944.851} C_VEL
LIN {X 0,Y 284.284,Z 219.073,A -85,B 0,C 180,E1 -16948.016,E2 -16948.016} C_VEL
LIN {X 0,Y 284.287,Z 219.07,A -85,B 0,C 180,E1 -16951.276,E2 -16951.276} C_VEL
LIN {X 0,Y 284.339,Z 219.067,A -85,B 0,C 180,E1 -16955.347,E2 -16955.347} C_VEL
LIN {X 0,Y 284.3,Z 219.07,A -85,B 0,C 180,E1 -16958.171,E2 -16958.171} C_VEL
LIN {X 0,Y 284.239,Z 219.078,A -85,B 0,C 180,E1 -16962.117,E2 -16962.117} C_VEL
LIN {X 0,Y 284.24,Z 219.077,A -85,B 0,C 180,E1 -16966.186,E2 -16966.186} C_VEL
LIN {X 0,Y 284.285,Z 219.072,A -85,B 0,C 180,E1 -16970.029,E2 -16970.029} C_VEL
LIN {X 0,Y 284.337,Z 219.067,A -85,B 0,C 180,E1 -16973.614,E2 -16973.614} C_VEL
LIN {X 0,Y 284.386,Z 219.179,A -85,B 0,C 180,E1 -16974.835,E2 -16974.835} C_VEL
LIN {X 0,Y 287.162,Z 232.205,A -85,B 0,C 180,E1 -16978.659,E2 -16978.659} C_VEL
LIN {X 0,Y 289.09,Z 241.676,A -85,B 0,C 180,E1 -16981.329,E2 -16981.329} C_VEL
LIN {X 0,Y 289.149,Z 244.593,A -85,B 0,C 180,E1 -16982.102,E2 -16982.102} C_VEL
LIN {X 0,Y 288.181,Z 251.597,A -85,B 0,C 180,E1 -16983.888,E2 -16983.888} C_VEL
LIN {X 0,Y 293.831,Z 302.082,A -85,B 0,C 180,E1 -16985.815,E2 -16985.815} C_VEL
LIN {X 0,Y 292.08,Z 361.945,A -85,B 0,C 180,E1 -16987.543,E2 -16987.543} C_VEL
LIN {X 0,Y 291.143,Z 375.611,A -85,B 0,C 180,E1 -16988.214,E2 -16988.214} C_VEL
LIN {X 0,Y 290.09,Z 387.544,A -85,B 0,C 180,E1 -16989.062,E2 -16989.062} C_VEL
LIN {X 0,Y 288.65,Z 400.022,A -85,B 0,C 180,E1 -16990.255,E2 -16990.255} C_VEL
LIN {X 0,Y 287.304,Z 411.278,A -85,B 0,C 180,E1 -16991.642,E2 -16991.642} C_VEL
LIN {X 0,Y 285.917,Z 421.81,A -85,B 0,C 180,E1 -16993.283,E2 -16993.283} C_VEL
LIN {X 0,Y 285.046,Z 428.974,A -85,B 0,C 180,E1 -16994.63,E2 -16994.63} C_VEL
LIN {X 0,Y 284.007,Z 438.247,A -85,B 0,C 180,E1 -16996.767,E2 -16996.767} C_VEL
LIN {X 0,Y 283.173,Z 445.682,A -85,B 0,C 180,E1 -16998.91,E2 -16998.91} C_VEL
LIN {X 0,Y 282.867,Z 450.7,A -85,B 0,C 180,E1 -17000.706,E2 -17000.706} C_VEL
LIN {X 0,Y 282.704,Z 455.531,A -85,B 0,C 180,E1 -17002.859,E2 -17002.859} C_VEL
LIN {X 0,Y 282.702,Z 459.165,A -85,B 0,C 180,E1 -17005.008,E2 -17005.008} C_VEL
LIN {X 0,Y 282.754,Z 461.703,A -85,B 0,C 180,E1 -17007.15,E2 -17007.15} C_VEL
LIN {X 0,Y 282.944,Z 462.857,A -85,B 0,C 180,E1 -17008.576,E2 -17008.576} C_VEL
LIN {X 0,Y 282.976,Z 463.519,A -85,B 0,C 180,E1 -17010,E2 -17010} C_VEL
LIN {X 0,Y 282.884,Z 463.753,A -85,B 0,C 180,E1 -17011.423,E2 -17011.423} C_VEL
LIN {X 0,Y 282.636,Z 463.566,A -85,B 0,C 180,E1 -17012.85,E2 -17012.85} C_VEL
LIN {X 0,Y 282.563,Z 462.976,A -85,B 0,C 180,E1 -17014.279,E2 -17014.279} C_VEL
LIN {X 0,Y 282.483,Z 461.931,A -85,B 0,C 180,E1 -17015.711,E2 -17015.711} C_VEL
LIN {X 0,Y 282.542,Z 460.483,A -85,B 0,C 180,E1 -17017.144,E2 -17017.144} C_VEL
LIN {X 0,Y 282.823,Z 457.501,A -85,B 0,C 180,E1 -17019.295,E2 -17019.295} C_VEL
LIN {X 0,Y 283.318,Z 453.48,A -85,B 0,C 180,E1 -17021.446,E2 -17021.446} C_VEL
LIN {X 0,Y 284.397,Z 448.349,A -85,B 0,C 180,E1 -17023.577,E2 -17023.577} C_VEL
LIN {X 0,Y 285.992,Z 440.941,A -85,B 0,C 180,E1 -17026.005,E2 -17026.005} C_VEL
LIN {X 0,Y 287.778,Z 432.62,A -85,B 0,C 180,E1 -17028.141,E2 -17028.141} C_VEL
LIN {X 0,Y 289.703,Z 424.358,A -85,B 0,C 180,E1 -17029.854,E2 -17029.854} C_VEL
LIN {X 0,Y 291.971,Z 414.362,A -85,B 0,C 180,E1 -17031.535,E2 -17031.535} C_VEL
LIN {X 0,Y 294.214,Z 403.31,A -85,B 0,C 180,E1 -17033.026,E2 -17033.026} C_VEL
LIN {X 0,Y 296.522,Z 390.924,A -85,B 0,C 180,E1 -17034.318,E2 -17034.318} C_VEL
LIN {X 0,Y 298.581,Z 377.893,A -85,B 0,C 180,E1 -17035.347,E2 -17035.347} C_VEL
LIN {X 0,Y 300.185,Z 364.671,A -85,B 0,C 180,E1 -17036.085,E2 -17036.085} C_VEL
LIN {X 0,Y 301.222,Z 350.898,A -85,B 0,C 180,E1 -17036.598,E2 -17036.598} C_VEL
LIN {X 0,Y 303.309,Z 303.646,A -85,B 0,C 180,E1 -17037.97,E2 -17037.97} C_VEL
LIN {X 0,Y 301.149,Z 283.239,A -85,B 0,C 180,E1 -17039.001,E2 -17039.001} C_VEL
LIN {X 0,Y 298.077,Z 264.009,A -85,B 0,C 180,E1 -17040.185,E2 -17040.185} C_VEL
LIN {X 0,Y 296.027,Z 255.04,A -85,B 0,C 180,E1 -17040.85,E2 -17040.85} C_VEL
LIN {X 0,Y 292.392,Z 247.365,A -85,B 0,C 180,E1 -17041.759,E2 -17041.759} C_VEL
LIN {X 0,Y 291.464,Z 245.022,A -85,B 0,C 180,E1 -17042.038,E2 -17042.038} C_VEL
LIN {X 0,Y 289.522,Z 236.492,A -85,B 0,C 180,E1 -17044.872,E2 -17044.872} C_VEL
LIN {X 0,Y 287.378,Z 228.775,A -85,B 0,C 180,E1 -17047.69,E2 -17047.69} C_VEL
LIN {X 0,Y 284.248,Z 219.076,A -85,B 0,C 180,E1 -17051.754,E2 -17051.754} C_VEL
LIN {X 0,Y 284.234,Z 219.076,A -85,B 0,C 180,E1 -17055.812,E2 -17055.812} C_VEL
LIN {X 0,Y 284.282,Z 219.069,A -85,B 0,C 180,E1 -17060.029,E2 -17060.029} C_VEL
LIN {X 0,Y 284.326,Z 219.069,A -85,B 0,C 180,E1 -17063.613,E2 -17063.613} C_VEL
LIN {X 0,Y 284.306,Z 219.067,A -85,B 0,C 180,E1 -17067.19,E2 -17067.19} C_VEL
LIN {X 0,Y 284.34,Z 219.06,A -85,B 0,C 180,E1 -17070.374,E2 -17070.374} C_VEL
LIN {X 0,Y 284.313,Z 219.063,A -85,B 0,C 180,E1 -17073.58,E2 -17073.58} C_VEL
LIN {X 0,Y 284.33,Z 219.062,A -85,B 0,C 180,E1 -17076.704,E2 -17076.704} C_VEL
LIN {X 0,Y 284.376,Z 219.056,A -85,B 0,C 180,E1 -17079.904,E2 -17079.904} C_VEL
LIN {X 0,Y 284.454,Z 219.05,A -85,B 0,C 180,E1 -17084.487,E2 -17084.487} C_VEL
LIN {X 0,Y 284.487,Z 219.042,A -85,B 0,C 180,E1 -17088.601,E2 -17088.601} C_VEL
LIN {X 0,Y 284.639,Z 219.025,A -85,B 0,C 180,E1 -17091.48,E2 -17091.48} C_VEL
LIN {X 0,Y 284.596,Z 219.032,A -85,B 0,C 180,E1 -17094.331,E2 -17094.331} C_VEL
LIN {X 0,Y 284.854,Z 218.999,A -85,B 0,C 180,E1 -17098.586,E2 -17098.586} C_VEL
LIN {X 0,Y 284.854,Z 219.003,A -85,B 0,C 180,E1 -17101.414,E2 -17101.414} C_VEL
LIN {X 0,Y 284.536,Z 219.042,A -85,B 0,C 180,E1 -17104.826,E2 -17104.826} C_VEL
LIN {X 0,Y 285.459,Z 221.767,A -85,B 0,C 180,E1 -17105.142,E2 -17105.142} C_VEL
LIN {X 0,Y 287.659,Z 224.403,A -85,B 0,C 180,E1 -17105.687,E2 -17105.687} C_VEL
LIN {X 0,Y 289.863,Z 227.763,A -85,B 0,C 180,E1 -17106.239,E2 -17106.239} C_VEL
LIN {X 0,Y 295.778,Z 237.577,A -85,B 0,C 180,E1 -17107.681,E2 -17107.681} C_VEL
LIN {X 0,Y 302.618,Z 250.124,A -85,B 0,C 180,E1 -17109.236,E2 -17109.236} C_VEL
LIN {X 0,Y 305.35,Z 255.884,A -85,B 0,C 180,E1 -17109.856,E2 -17109.856} C_VEL
LIN {X 0,Y 302.085,Z 322.365,A -85,B 0,C 180,E1 -17111.803,E2 -17111.803} C_VEL
LIN {X 0,Y 301.172,Z 335.641,A -85,B 0,C 180,E1 -17112.466,E2 -17112.466} C_VEL
LIN {X 0,Y 299.837,Z 348.543,A -85,B 0,C 180,E1 -17113.383,E2 -17113.383} C_VEL
LIN {X 0,Y 298.184,Z 360.129,A -85,B 0,C 180,E1 -17114.485,E2 -17114.485} C_VEL
LIN {X 0,Y 296.36,Z 371.102,A -85,B 0,C 180,E1 -17115.826,E2 -17115.826} C_VEL
LIN {X 0,Y 294.422,Z 380.776,A -85,B 0,C 180,E1 -17117.289,E2 -17117.289} C_VEL
LIN {X 0,Y 292.574,Z 389.503,A -85,B 0,C 180,E1 -17118.922,E2 -17118.922} C_VEL
LIN {X 0,Y 290.514,Z 398.063,A -85,B 0,C 180,E1 -17120.911,E2 -17120.911} C_VEL
LIN {X 0,Y 288.685,Z 405.006,A -85,B 0,C 180,E1 -17122.924,E2 -17122.924} C_VEL
LIN {X 0,Y 287.089,Z 410.861,A -85,B 0,C 180,E1 -17125.074,E2 -17125.074} C_VEL
LIN {X 0,Y 285.964,Z 414.79,A -85,B 0,C 180,E1 -17126.918,E2 -17126.918} C_VEL
LIN {X 0,Y 284.627,Z 419.026,A -85,B 0,C 180,E1 -17129.593,E2 -17129.593} C_VEL
LIN {X 0,Y 283.974,Z 420.879,A -85,B 0,C 180,E1 -17131.314,E2 -17131.314} C_VEL
LIN {X 0,Y 283.425,Z 422.137,A -85,B 0,C 180,E1 -17133.061,E2 -17133.061} C_VEL
LIN {X 0,Y 283.013,Z 422.813,A -85,B 0,C 180,E1 -17134.968,E2 -17134.968} C_VEL
LIN {X 0,Y 282.726,Z 422.62,A -85,B 0,C 180,E1 -17137.302,E2 -17137.302} C_VEL
LIN {X 0,Y 282.658,Z 421.376,A -85,B 0,C 180,E1 -17139.576,E2 -17139.576} C_VEL
LIN {X 0,Y 282.917,Z 418.695,A -85,B 0,C 180,E1 -17142.122,E2 -17142.122} C_VEL
LIN {X 0,Y 283.268,Z 415.84,A -85,B 0,C 180,E1 -17144.003,E2 -17144.003} C_VEL
LIN {X 0,Y 283.759,Z 411.66,A -85,B 0,C 180,E1 -17146.093,E2 -17146.093} C_VEL
LIN {X 0,Y 284.485,Z 405.394,A -85,B 0,C 180,E1 -17148.495,E2 -17148.495} C_VEL
LIN {X 0,Y 285.332,Z 398.458,A -85,B 0,C 180,E1 -17150.595,E2 -17150.595} C_VEL
LIN {X 0,Y 286.46,Z 390.265,A -85,B 0,C 180,E1 -17152.59,E2 -17152.59} C_VEL
LIN {X 0,Y 287.676,Z 380.295,A -85,B 0,C 180,E1 -17154.535,E2 -17154.535} C_VEL
LIN {X 0,Y 288.886,Z 369.794,A -85,B 0,C 180,E1 -17156.186,E2 -17156.186} C_VEL
LIN {X 0,Y 290.091,Z 358.547,A -85,B 0,C 180,E1 -17157.587,E2 -17157.587} C_VEL
LIN {X 0,Y 291.289,Z 345.463,A -85,B 0,C 180,E1 -17158.854,E2 -17158.854} C_VEL
LIN {X 0,Y 292.158,Z 332.337,A -85,B 0,C 180,E1 -17159.787,E2 -17159.787} C_VEL
LIN {X 0,Y 292.712,Z 319.634,A -85,B 0,C 180,E1 -17160.416,E2 -17160.416} C_VEL
LIN {X 0,Y 293.911,Z 279.295,A -85,B 0,C 180,E1 -17161.588,E2 -17161.588} C_VEL
LIN {X 0,Y 294.868,Z 246.214,A -85,B 0,C 180,E1 -17162.52,E2 -17162.52} C_VEL
LIN {X 0,Y 284.444,Z 219.452,A -85,B 0,C 180,E1 -17164.086,E2 -17164.086} C_VEL
LIN {X 0,Y 284.4,Z 219.058,A -85,B 0,C 180,E1 -17164.18,E2 -17164.18} C_VEL
LIN {X 0,Y 284.315,Z 219.068,A -85,B 0,C 180,E1 -17168.236,E2 -17168.236} C_VEL
LIN {X 0,Y 284.376,Z 219.062,A -85,B 0,C 180,E1 -17171.26,E2 -17171.26} C_VEL
LIN {X 0,Y 284.464,Z 219.049,A -85,B 0,C 180,E1 -17175.697,E2 -17175.697} C_VEL
LIN {X 0,Y 284.515,Z 219.043,A -85,B 0,C 180,E1 -17180.043,E2 -17180.043} C_VEL
LIN {X 0,Y 284.647,Z 219.029,A -85,B 0,C 180,E1 -17182.909,E2 -17182.909} C_VEL
LIN {X 0,Y 284.853,Z 219.004,A -85,B 0,C 180,E1 -17188.587,E2 -17188.587} C_VEL
LIN {X 0,Y 284.852,Z 219,A -85,B 0,C 180,E1 -17191.414,E2 -17191.414} C_VEL
LIN {X 0,Y 284.654,Z 219.025,A -85,B 0,C 180,E1 -17197.092,E2 -17197.092} C_VEL
LIN {X 0,Y 284.519,Z 219.044,A -85,B 0,C 180,E1 -17199.957,E2 -17199.957} C_VEL
LIN {X 0,Y 284.483,Z 219.05,A -85,B 0,C 180,E1 -17204.303,E2 -17204.303} C_VEL
LIN {X 0,Y 284.425,Z 219.053,A -85,B 0,C 180,E1 -17207.249,E2 -17207.249} C_VEL
LIN {X 0,Y 284.379,Z 219.058,A -85,B 0,C 180,E1 -17210.243,E2 -17210.243} C_VEL
LIN {X 0,Y 284.327,Z 219.066,A -85,B 0,C 180,E1 -17213.856,E2 -17213.856} C_VEL
LIN {X 0,Y 284.29,Z 219.074,A -85,B 0,C 180,E1 -17218.016,E2 -17218.016} C_VEL
LIN {X 0,Y 284.288,Z 219.071,A -85,B 0,C 180,E1 -17221.276,E2 -17221.276} C_VEL
LIN {X 0,Y 284.338,Z 219.063,A -85,B 0,C 180,E1 -17225.347,E2 -17225.347} C_VEL
LIN {X 0,Y 284.301,Z 219.062,A -85,B 0,C 180,E1 -17228.171,E2 -17228.171} C_VEL
LIN {X 0,Y 284.253,Z 219.073,A -85,B 0,C 180,E1 -17232.121,E2 -17232.121} C_VEL
LIN {X 0,Y 284.257,Z 219.074,A -85,B 0,C 180,E1 -17236.19,E2 -17236.19} C_VEL
LIN {X 0,Y 284.285,Z 219.07,A -85,B 0,C 180,E1 -17240.03,E2 -17240.03} C_VEL
LIN {X 0,Y 284.33,Z 219.065,A -85,B 0,C 180,E1 -17243.614,E2 -17243.614} C_VEL
LIN {X 0,Y 284.308,Z 219.072,A -85,B 0,C 180,E1 -17247.191,E2 -17247.191} C_VEL
LIN {X 0,Y 284.339,Z 219.064,A -85,B 0,C 180,E1 -17250.374,E2 -17250.374} C_VEL
LIN {X 0,Y 284.308,Z 219.066,A -85,B 0,C 180,E1 -17253.58,E2 -17253.58} C_VEL
LIN {X 0,Y 284.331,Z 219.066,A -85,B 0,C 180,E1 -17256.704,E2 -17256.704} C_VEL
LIN {X 0,Y 284.379,Z 219.059,A -85,B 0,C 180,E1 -17259.905,E2 -17259.905} C_VEL
LIN {X 0,Y 284.45,Z 219.051,A -85,B 0,C 180,E1 -17264.492,E2 -17264.492} C_VEL
LIN {X 0,Y 284.442,Z 219.049,A -85,B 0,C 180,E1 -17264.962,E2 -17264.962} C_VEL
LIN {X 0,Y 283.791,Z 219.132,A -85,B 0,C 180,E1 -17266.143,E2 -17266.143} C_VEL
LIN {X 0,Y 280.986,Z 219.477,A -85,B 0,C 180,E1 -17268.068,E2 -17268.068} C_VEL
LIN {X 0,Y 278.622,Z 219.771,A -85,B 0,C 180,E1 -17269.632,E2 -17269.632} C_VEL
LIN {X 0,Y 277.637,Z 219.893,A -85,B 0,C 180,E1 -17270.843,E2 -17270.843} C_VEL
LIN {X 0,Y 277.572,Z 219.899,A -85,B 0,C 180,E1 -17271.253,E2 -17271.253} C_VEL
LIN {X 0,Y 277.546,Z 219.908,A -85,B 0,C 180,E1 -17274.187,E2 -17274.187} C_VEL
LIN {X 0,Y 277.812,Z 219.88,A -85,B 0,C 180,E1 -17278.55,E2 -17278.55} C_VEL
LIN {X 0,Y 277.814,Z 219.877,A -85,B 0,C 180,E1 -17281.45,E2 -17281.45} C_VEL
LIN {X 0,Y 277.604,Z 219.897,A -85,B 0,C 180,E1 -17287.272,E2 -17287.272} C_VEL
LIN {X 0,Y 277.463,Z 219.922,A -85,B 0,C 180,E1 -17290.213,E2 -17290.213} C_VEL
LIN {X 0,Y 277.39,Z 219.931,A -85,B 0,C 180,E1 -17294.677,E2 -17294.677} C_VEL
LIN {X 0,Y 277.325,Z 219.937,A -85,B 0,C 180,E1 -17299.235,E2 -17299.235} C_VEL
LIN {X 0,Y 277.263,Z 219.95,A -85,B 0,C 180,E1 -17303.927,E2 -17303.927} C_VEL
LIN {X 0,Y 277.27,Z 219.949,A -85,B 0,C 180,E1 -17307.482,E2 -17307.482} C_VEL
LIN {X 0,Y 277.25,Z 219.945,A -85,B 0,C 180,E1 -17310.473,E2 -17310.473} C_VEL
LIN {X 0,Y 277.248,Z 219.949,A -85,B 0,C 180,E1 -17313.896,E2 -17313.896} C_VEL
LIN {X 0,Y 277.257,Z 219.951,A -85,B 0,C 180,E1 -17317.471,E2 -17317.471} C_VEL
LIN {X 0,Y 277.186,Z 219.96,A -85,B 0,C 180,E1 -17321.241,E2 -17321.241} C_VEL
LIN {X 0,Y 277.176,Z 219.961,A -85,B 0,C 180,E1 -17325.232,E2 -17325.232} C_VEL
LIN {X 0,Y 277.186,Z 219.957,A -85,B 0,C 180,E1 -17328.759,E2 -17328.759} C_VEL
LIN {X 0,Y 277.264,Z 219.948,A -85,B 0,C 180,E1 -17332.53,E2 -17332.53} C_VEL
LIN {X 0,Y 277.343,Z 220.098,A -85,B 0,C 180,E1 -17334.461,E2 -17334.461} C_VEL
LIN {X 0,Y 279.991,Z 232.451,A -85,B 0,C 180,E1 -17338.189,E2 -17338.189} C_VEL
LIN {X 0,Y 282.164,Z 243.192,A -85,B 0,C 180,E1 -17341.295,E2 -17341.295} C_VEL
LIN {X 0,Y 282.034,Z 246.364,A -85,B 0,C 180,E1 -17342.145,E2 -17342.145} C_VEL
LIN {X 0,Y 281.34,Z 251.128,A -85,B 0,C 180,E1 -17343.387,E2 -17343.387} C_VEL
LIN {X 0,Y 287.066,Z 302.608,A -85,B 0,C 180,E1 -17345.405,E2 -17345.405} C_VEL
LIN {X 0,Y 285.305,Z 360.758,A -85,B 0,C 180,E1 -17347.123,E2 -17347.123} C_VEL
LIN {X 0,Y 284.359,Z 374.603,A -85,B 0,C 180,E1 -17347.809,E2 -17347.809} C_VEL
LIN {X 0,Y 283.213,Z 387.175,A -85,B 0,C 180,E1 -17348.72,E2 -17348.72} C_VEL
LIN {X 0,Y 281.739,Z 399.61,A -85,B 0,C 180,E1 -17349.94,E2 -17349.94} C_VEL
LIN {X 0,Y 280.36,Z 410.844,A -85,B 0,C 180,E1 -17351.36,E2 -17351.36} C_VEL
LIN {X 0,Y 279.143,Z 419.973,A -85,B 0,C 180,E1 -17352.793,E2 -17352.793} C_VEL
LIN {X 0,Y 278.076,Z 427.605,A -85,B 0,C 180,E1 -17354.235,E2 -17354.235} C_VEL
LIN {X 0,Y 277.167,Z 435.668,A -85,B 0,C 180,E1 -17356.061,E2 -17356.061} C_VEL
LIN {X 0,Y 276.443,Z 442.324,A -85,B 0,C 180,E1 -17357.892,E2 -17357.892} C_VEL
LIN {X 0,Y 275.929,Z 447.826,A -85,B 0,C 180,E1 -17359.729,E2 -17359.729} C_VEL
LIN {X 0,Y 275.667,Z 453.188,A -85,B 0,C 180,E1 -17361.939,E2 -17361.939} C_VEL
LIN {X 0,Y 275.659,Z 457.301,A -85,B 0,C 180,E1 -17364.146,E2 -17364.146} C_VEL
LIN {X 0,Y 275.646,Z 459.38,A -85,B 0,C 180,E1 -17365.613,E2 -17365.613} C_VEL
LIN {X 0,Y 275.671,Z 461,A -85,B 0,C 180,E1 -17367.077,E2 -17367.077} C_VEL
LIN {X 0,Y 275.865,Z 462.202,A -85,B 0,C 180,E1 -17368.54,E2 -17368.54} C_VEL
LIN {X 0,Y 275.921,Z 462.931,A -85,B 0,C 180,E1 -17370,E2 -17370} C_VEL
LIN {X 0,Y 275.788,Z 463.198,A -85,B 0,C 180,E1 -17371.46,E2 -17371.46} C_VEL
LIN {X 0,Y 275.471,Z 462.499,A -85,B 0,C 180,E1 -17374.389,E2 -17374.389} C_VEL
LIN {X 0,Y 275.39,Z 461.513,A -85,B 0,C 180,E1 -17375.859,E2 -17375.859} C_VEL
LIN {X 0,Y 275.472,Z 460.097,A -85,B 0,C 180,E1 -17377.328,E2 -17377.328} C_VEL
LIN {X 0,Y 275.756,Z 457.192,A -85,B 0,C 180,E1 -17379.535,E2 -17379.535} C_VEL
LIN {X 0,Y 276.318,Z 453.272,A -85,B 0,C 180,E1 -17381.74,E2 -17381.74} C_VEL
LIN {X 0,Y 277.475,Z 448.244,A -85,B 0,C 180,E1 -17383.923,E2 -17383.923} C_VEL
LIN {X 0,Y 278.894,Z 441.962,A -85,B 0,C 180,E1 -17386.092,E2 -17386.092} C_VEL
LIN {X 0,Y 280.661,Z 434.217,A -85,B 0,C 180,E1 -17388.24,E2 -17388.24} C_VEL
LIN {X 0,Y 282.6,Z 426.388,A -85,B 0,C 180,E1 -17389.995,E2 -17389.995} C_VEL
LIN {X 0,Y 284.913,Z 417.027,A -85,B 0,C 180,E1 -17391.716,E2 -17391.716} C_VEL
LIN {X 0,Y 287.184,Z 406.735,A -85,B 0,C 180,E1 -17393.241,E2 -17393.241} C_VEL
LIN {X 0,Y 289.526,Z 395.466,A -85,B 0,C 180,E1 -17394.563,E2 -17394.563} C_VEL
LIN {X 0,Y 291.796,Z 382.98,A -85,B 0,C 180,E1 -17395.692,E2 -17395.692} C_VEL
LIN {X 0,Y 293.644,Z 370.44,A -85,B 0,C 180,E1 -17396.52,E2 -17396.52} C_VEL
LIN {X 0,Y 294.943,Z 356.955,A -85,B 0,C 180,E1 -17397.16,E2 -17397.16} C_VEL
LIN {X 0,Y 297.546,Z 304.67,A -85,B 0,C 180,E1 -17398.731,E2 -17398.731} C_VEL
LIN {X 0,Y 295.518,Z 284.786,A -85,B 0,C 180,E1 -17399.785,E2 -17399.785} C_VEL
LIN {X 0,Y 292.698,Z 266.502,A -85,B 0,C 180,E1 -17400.94,E2 -17400.94} C_VEL
LIN {X 0,Y 290.938,Z 258.543,A -85,B 0,C 180,E1 -17401.553,E2 -17401.553} C_VEL
LIN {X 0,Y 286.4,Z 248.788,A -85,B 0,C 180,E1 -17402.765,E2 -17402.765} C_VEL
LIN {X 0,Y 284.239,Z 244.123,A -85,B 0,C 180,E1 -17403.401,E2 -17403.401} C_VEL
LIN {X 0,Y 281.924,Z 234.806,A -85,B 0,C 180,E1 -17406.747,E2 -17406.747} C_VEL
LIN {X 0,Y 279.485,Z 226.985,A -85,B 0,C 180,E1 -17409.918,E2 -17409.918} C_VEL
LIN {X 0,Y 277.191,Z 219.951,A -85,B 0,C 180,E1 -17413.201,E2 -17413.201} C_VEL
LIN {X 0,Y 277.192,Z 219.951,A -85,B 0,C 180,E1 -17417.33,E2 -17417.33} C_VEL
LIN {X 0,Y 277.255,Z 219.946,A -85,B 0,C 180,E1 -17421.795,E2 -17421.795} C_VEL
LIN {X 0,Y 277.279,Z 219.943,A -85,B 0,C 180,E1 -17424.34,E2 -17424.34} C_VEL
LIN {X 0,Y 277.24,Z 219.945,A -85,B 0,C 180,E1 -17427.836,E2 -17427.836} C_VEL
LIN {X 0,Y 277.243,Z 219.946,A -85,B 0,C 180,E1 -17431.207,E2 -17431.207} C_VEL
LIN {X 0,Y 277.253,Z 219.948,A -85,B 0,C 180,E1 -17434.473,E2 -17434.473} C_VEL
LIN {X 0,Y 277.265,Z 219.947,A -85,B 0,C 180,E1 -17437.653,E2 -17437.653} C_VEL
LIN {X 0,Y 277.329,Z 219.94,A -85,B 0,C 180,E1 -17440.765,E2 -17440.765} C_VEL
LIN {X 0,Y 277.414,Z 219.922,A -85,B 0,C 180,E1 -17445.325,E2 -17445.325} C_VEL
LIN {X 0,Y 277.461,Z 219.924,A -85,B 0,C 180,E1 -17449.787,E2 -17449.787} C_VEL
LIN {X 0,Y 277.641,Z 219.902,A -85,B 0,C 180,E1 -17452.729,E2 -17452.729} C_VEL
LIN {X 0,Y 277.82,Z 219.876,A -85,B 0,C 180,E1 -17458.55,E2 -17458.55} C_VEL
LIN {X 0,Y 277.82,Z 219.88,A -85,B 0,C 180,E1 -17461.449,E2 -17461.449} C_VEL
LIN {X 0,Y 277.588,Z 219.943,A -85,B 0,C 180,E1 -17463.402,E2 -17463.402} C_VEL
LIN {X 0,Y 278.555,Z 222.773,A -85,B 0,C 180,E1 -17463.752,E2 -17463.752} C_VEL
LIN {X 0,Y 280.621,Z 225.199,A -85,B 0,C 180,E1 -17464.309,E2 -17464.309} C_VEL
LIN {X 0,Y 282.53,Z 228.335,A -85,B 0,C 180,E1 -17464.851,E2 -17464.851} C_VEL
LIN {X 0,Y 283.924,Z 230.224,A -85,B 0,C 180,E1 -17465.217,E2 -17465.217} C_VEL
LIN {X 0,Y 288.736,Z 237.748,A -85,B 0,C 180,E1 -17466.452,E2 -17466.452} C_VEL
LIN {X 0,Y 295.675,Z 250.184,A -85,B 0,C 180,E1 -17468.156,E2 -17468.156} C_VEL
LIN {X 0,Y 299.647,Z 258.173,A -85,B 0,C 180,E1 -17469.087,E2 -17469.087} C_VEL
LIN {X 0,Y 296.198,Z 323.586,A -85,B 0,C 180,E1 -17471.069,E2 -17471.069} C_VEL
LIN {X 0,Y 295.25,Z 336.599,A -85,B 0,C 180,E1 -17471.742,E2 -17471.742} C_VEL
LIN {X 0,Y 293.821,Z 349.615,A -85,B 0,C 180,E1 -17472.695,E2 -17472.695} C_VEL
LIN {X 0,Y 291.911,Z 362.155,A -85,B 0,C 180,E1 -17473.931,E2 -17473.931} C_VEL
LIN {X 0,Y 290.081,Z 372.481,A -85,B 0,C 180,E1 -17475.242,E2 -17475.242} C_VEL
LIN {X 0,Y 287.876,Z 382.685,A -85,B 0,C 180,E1 -17476.852,E2 -17476.852} C_VEL
LIN {X 0,Y 285.793,Z 391.698,A -85,B 0,C 180,E1 -17478.644,E2 -17478.644} C_VEL
LIN {X 0,Y 283.678,Z 399.927,A -85,B 0,C 180,E1 -17480.673,E2 -17480.673} C_VEL
LIN {X 0,Y 281.502,Z 407.506,A -85,B 0,C 180,E1 -17483.05,E2 -17483.05} C_VEL
LIN {X 0,Y 279.873,Z 413.05,A -85,B 0,C 180,E1 -17485.311,E2 -17485.311} C_VEL
LIN {X 0,Y 278.371,Z 417.828,A -85,B 0,C 180,E1 -17487.916,E2 -17487.916} C_VEL
LIN {X 0,Y 277.226,Z 420.977,A -85,B 0,C 180,E1 -17490.466,E2 -17490.466} C_VEL
LIN {X 0,Y 276.395,Z 422.784,A -85,B 0,C 180,E1 -17492.955,E2 -17492.955} C_VEL
LIN {X 0,Y 275.802,Z 423.406,A -85,B 0,C 180,E1 -17495.88,E2 -17495.88} C_VEL
LIN {X 0,Y 275.607,Z 422.902,A -85,B 0,C 180,E1 -17497.768,E2 -17497.768} C_VEL
LIN {X 0,Y 275.612,Z 421.367,A -85,B 0,C 180,E1 -17500.095,E2 -17500.095} C_VEL
LIN {X 0,Y 275.891,Z 418.816,A -85,B 0,C 180,E1 -17502.376,E2 -17502.376} C_VEL
LIN {X 0,Y 276.286,Z 415.307,A -85,B 0,C 180,E1 -17504.582,E2 -17504.582} C_VEL
LIN {X 0,Y 276.818,Z 410.813,A -85,B 0,C 180,E1 -17506.726,E2 -17506.726} C_VEL
LIN {X 0,Y 277.495,Z 405.276,A -85,B 0,C 180,E1 -17508.816,E2 -17508.816} C_VEL
LIN {X 0,Y 278.345,Z 398.571,A -85,B 0,C 180,E1 -17510.859,E2 -17510.859} C_VEL
LIN {X 0,Y 279.508,Z 390.344,A -85,B 0,C 180,E1 -17512.882,E2 -17512.882} C_VEL
LIN {X 0,Y 280.748,Z 380.428,A -85,B 0,C 180,E1 -17514.847,E2 -17514.847} C_VEL
LIN {X 0,Y 281.953,Z 370.324,A -85,B 0,C 180,E1 -17516.466,E2 -17516.466} C_VEL
LIN {X 0,Y 283.108,Z 359.741,A -85,B 0,C 180,E1 -17517.827,E2 -17517.827} C_VEL
LIN {X 0,Y 284.348,Z 346.968,A -85,B 0,C 180,E1 -17519.109,E2 -17519.109} C_VEL
LIN {X 0,Y 285.226,Z 334.967,A -85,B 0,C 180,E1 -17520.023,E2 -17520.023} C_VEL
LIN {X 0,Y 285.782,Z 322.45,A -85,B 0,C 180,E1 -17520.703,E2 -17520.703} C_VEL
LIN {X 0,Y 286.422,Z 302.83,A -85,B 0,C 180,E1 -17521.34,E2 -17521.34} C_VEL
LIN {X 0,Y 288.106,Z 247.783,A -85,B 0,C 180,E1 -17522.929,E2 -17522.929} C_VEL
LIN {X 0,Y 278.011,Z 222.212,A -85,B 0,C 180,E1 -17524.486,E2 -17524.486} C_VEL
LIN {X 0,Y 277.327,Z 219.941,A -85,B 0,C 180,E1 -17524.639,E2 -17524.639} C_VEL
LIN {X 0,Y 277.285,Z 219.946,A -85,B 0,C 180,E1 -17529.217,E2 -17529.217} C_VEL
LIN {X 0,Y 277.331,Z 219.938,A -85,B 0,C 180,E1 -17532.296,E2 -17532.296} C_VEL
LIN {X 0,Y 277.41,Z 219.929,A -85,B 0,C 180,E1 -17535.325,E2 -17535.325} C_VEL
LIN {X 0,Y 277.458,Z 219.922,A -85,B 0,C 180,E1 -17539.787,E2 -17539.787} C_VEL
LIN {X 0,Y 277.605,Z 219.907,A -85,B 0,C 180,E1 -17542.728,E2 -17542.728} C_VEL
LIN {X 0,Y 277.819,Z 219.88,A -85,B 0,C 180,E1 -17548.551,E2 -17548.551} C_VEL
LIN {X 0,Y 277.817,Z 219.876,A -85,B 0,C 180,E1 -17551.45,E2 -17551.45} C_VEL
LIN {X 0,Y 277.612,Z 219.902,A -85,B 0,C 180,E1 -17557.272,E2 -17557.272} C_VEL
LIN {X 0,Y 277.462,Z 219.925,A -85,B 0,C 180,E1 -17560.213,E2 -17560.213} C_VEL
LIN {X 0,Y 277.436,Z 219.925,A -85,B 0,C 180,E1 -17564.674,E2 -17564.674} C_VEL
LIN {X 0,Y 277.344,Z 219.934,A -85,B 0,C 180,E1 -17569.234,E2 -17569.234} C_VEL
LIN {X 0,Y 277.288,Z 219.943,A -85,B 0,C 180,E1 -17573.925,E2 -17573.925} C_VEL
LIN {X 0,Y 277.276,Z 219.945,A -85,B 0,C 180,E1 -17577.485,E2 -17577.485} C_VEL
LIN {X 0,Y 277.249,Z 219.947,A -85,B 0,C 180,E1 -17580.473,E2 -17580.473} C_VEL
LIN {X 0,Y 277.247,Z 219.946,A -85,B 0,C 180,E1 -17583.896,E2 -17583.896} C_VEL
LIN {X 0,Y 277.256,Z 219.941,A -85,B 0,C 180,E1 -17587.472,E2 -17587.472} C_VEL
LIN {X 0,Y 277.203,Z 219.95,A -85,B 0,C 180,E1 -17591.238,E2 -17591.238} C_VEL
LIN {X 0,Y 277.203,Z 219.955,A -85,B 0,C 180,E1 -17595.227,E2 -17595.227} C_VEL
LIN {X 0,Y 277.199,Z 219.956,A -85,B 0,C 180,E1 -17599.519,E2 -17599.519} C_VEL
LIN {X 0,Y 277.262,Z 219.943,A -85,B 0,C 180,E1 -17602.53,E2 -17602.53} C_VEL
LIN {X 0,Y 277.249,Z 219.946,A -85,B 0,C 180,E1 -17606.105,E2 -17606.105} C_VEL
LIN {X 0,Y 277.264,Z 219.947,A -85,B 0,C 180,E1 -17609.539,E2 -17609.539} C_VEL
LIN {X 0,Y 277.294,Z 219.944,A -85,B 0,C 180,E1 -17612.857,E2 -17612.857} C_VEL
LIN {X 0,Y 277.285,Z 219.941,A -85,B 0,C 180,E1 -17616.076,E2 -17616.076} C_VEL
LIN {X 0,Y 277.328,Z 219.941,A -85,B 0,C 180,E1 -17620.765,E2 -17620.765} C_VEL
LIN {X 0,Y 277.413,Z 219.924,A -85,B 0,C 180,E1 -17625.325,E2 -17625.325} C_VEL
LIN {X 0,Y 277.46,Z 219.911,A -85,B 0,C 180,E1 -17629.787,E2 -17629.787} C_VEL
LIN {X 0,Y 277.572,Z 219.899,A -85,B 0,C 180,E1 -17631.253,E2 -17631.253} C_VEL
LIN {X 0,Y 276.937,Z 219.982,A -85,B 0,C 180,E1 -17632.463,E2 -17632.463} C_VEL
LIN {X 0,Y 274.08,Z 220.341,A -85,B 0,C 180,E1 -17634.433,E2 -17634.433} C_VEL
LIN {X 0,Y 271.679,Z 220.64,A -85,B 0,C 180,E1 -17636.035,E2 -17636.035} C_VEL
LIN {X 0,Y 270.712,Z 220.761,A -85,B 0,C 180,E1 -17637.277,E2 -17637.277} C_VEL
LIN {X 0,Y 270.669,Z 220.766,A -85,B 0,C 180,E1 -17637.697,E2 -17637.697} C_VEL
LIN {X 0,Y 270.778,Z 220.753,A -85,B 0,C 180,E1 -17641.487,E2 -17641.487} C_VEL
LIN {X 0,Y 270.565,Z 220.773,A -85,B 0,C 180,E1 -17647.463,E2 -17647.463} C_VEL
LIN {X 0,Y 270.414,Z 220.798,A -85,B 0,C 180,E1 -17650.482,E2 -17650.482} C_VEL
LIN {X 0,Y 270.355,Z 220.807,A -85,B 0,C 180,E1 -17655.068,E2 -17655.068} C_VEL
LIN {X 0,Y 270.262,Z 220.82,A -85,B 0,C 180,E1 -17659.759,E2 -17659.759} C_VEL
LIN {X 0,Y 270.182,Z 220.828,A -85,B 0,C 180,E1 -17664.595,E2 -17664.595} C_VEL
LIN {X 0,Y 270.199,Z 220.828,A -85,B 0,C 180,E1 -17667.917,E2 -17667.917} C_VEL
LIN {X 0,Y 270.176,Z 220.828,A -85,B 0,C 180,E1 -17671.349,E2 -17671.349} C_VEL
LIN {X 0,Y 270.201,Z 220.826,A -85,B 0,C 180,E1 -17674.906,E2 -17674.906} C_VEL
LIN {X 0,Y 270.2,Z 220.827,A -85,B 0,C 180,E1 -17678.71,E2 -17678.71} C_VEL
LIN {X 0,Y 270.15,Z 220.836,A -85,B 0,C 180,E1 -17683.245,E2 -17683.245} C_VEL
LIN {X 0,Y 270.153,Z 220.835,A -85,B 0,C 180,E1 -17687.437,E2 -17687.437} C_VEL
LIN {X 0,Y 270.21,Z 220.828,A -85,B 0,C 180,E1 -17691.374,E2 -17691.374} C_VEL
LIN {X 0,Y 270.246,Z 220.847,A -85,B 0,C 180,E1 -17694.024,E2 -17694.024} C_VEL
LIN {X 0,Y 273.102,Z 234.089,A -85,B 0,C 180,E1 -17698.128,E2 -17698.128} C_VEL
LIN {X 0,Y 275.039,Z 243.631,A -85,B 0,C 180,E1 -17700.954,E2 -17700.954} C_VEL
LIN {X 0,Y 275.129,Z 246.648,A -85,B 0,C 180,E1 -17701.798,E2 -17701.798} C_VEL
LIN {X 0,Y 274.538,Z 250.899,A -85,B 0,C 180,E1 -17702.877,E2 -17702.877} C_VEL
LIN {X 0,Y 280.229,Z 303.706,A -85,B 0,C 180,E1 -17705.004,E2 -17705.004} C_VEL
LIN {X 0,Y 278.454,Z 360.3,A -85,B 0,C 180,E1 -17706.724,E2 -17706.724} C_VEL
LIN {X 0,Y 277.595,Z 373.413,A -85,B 0,C 180,E1 -17707.386,E2 -17707.386} C_VEL
LIN {X 0,Y 276.347,Z 386.685,A -85,B 0,C 180,E1 -17708.36,E2 -17708.36} C_VEL
LIN {X 0,Y 274.837,Z 399.114,A -85,B 0,C 180,E1 -17709.609,E2 -17709.609} C_VEL
LIN {X 0,Y 273.423,Z 410.346,A -85,B 0,C 180,E1 -17711.064,E2 -17711.064} C_VEL
LIN {X 0,Y 271.964,Z 420.873,A -85,B 0,C 180,E1 -17712.789,E2 -17712.789} C_VEL
LIN {X 0,Y 270.981,Z 428.072,A -85,B 0,C 180,E1 -17714.213,E2 -17714.213} C_VEL
LIN {X 0,Y 269.916,Z 437.27,A -85,B 0,C 180,E1 -17716.447,E2 -17716.447} C_VEL
LIN {X 0,Y 269.043,Z 444.694,A -85,B 0,C 180,E1 -17718.701,E2 -17718.701} C_VEL
LIN {X 0,Y 268.67,Z 450.612,A -85,B 0,C 180,E1 -17720.97,E2 -17720.97} C_VEL
LIN {X 0,Y 268.57,Z 455.339,A -85,B 0,C 180,E1 -17723.312,E2 -17723.312} C_VEL
LIN {X 0,Y 268.587,Z 458.639,A -85,B 0,C 180,E1 -17725.497,E2 -17725.497} C_VEL
LIN {X 0,Y 268.589,Z 460.297,A -85,B 0,C 180,E1 -17727,E2 -17727} C_VEL
LIN {X 0,Y 268.789,Z 461.537,A -85,B 0,C 180,E1 -17728.501,E2 -17728.501} C_VEL
LIN {X 0,Y 268.866,Z 462.335,A -85,B 0,C 180,E1 -17730,E2 -17730} C_VEL
LIN {X 0,Y 268.694,Z 462.643,A -85,B 0,C 180,E1 -17731.498,E2 -17731.498} C_VEL
LIN {X 0,Y 268.382,Z 462.014,A -85,B 0,C 180,E1 -17734.505,E2 -17734.505} C_VEL
LIN {X 0,Y 268.303,Z 461.095,A -85,B 0,C 180,E1 -17736.014,E2 -17736.014} C_VEL
LIN {X 0,Y 268.385,Z 459.731,A -85,B 0,C 180,E1 -17737.523,E2 -17737.523} C_VEL
LIN {X 0,Y 268.695,Z 456.913,A -85,B 0,C 180,E1 -17739.788,E2 -17739.788} C_VEL
LIN {X 0,Y 269.327,Z 453.078,A -85,B 0,C 180,E1 -17742.049,E2 -17742.049} C_VEL
LIN {X 0,Y 270.567,Z 448.14,A -85,B 0,C 180,E1 -17744.286,E2 -17744.286} C_VEL
LIN {X 0,Y 272.425,Z 440.616,A -85,B 0,C 180,E1 -17746.93,E2 -17746.93} C_VEL
LIN {X 0,Y 274.292,Z 432.973,A -85,B 0,C 180,E1 -17749.067,E2 -17749.067} C_VEL
LIN {X 0,Y 276.411,Z 425.055,A -85,B 0,C 180,E1 -17750.852,E2 -17750.852} C_VEL
LIN {X 0,Y 279.141,Z 414.402,A -85,B 0,C 180,E1 -17752.774,E2 -17752.774} C_VEL
LIN {X 0,Y 281.579,Z 403.69,A -85,B 0,C 180,E1 -17754.319,E2 -17754.319} C_VEL
LIN {X 0,Y 284.094,Z 391.797,A -85,B 0,C 180,E1 -17755.653,E2 -17755.653} C_VEL
LIN {X 0,Y 286.495,Z 378.273,A -85,B 0,C 180,E1 -17756.792,E2 -17756.792} C_VEL
LIN {X 0,Y 288.311,Z 365.113,A -85,B 0,C 180,E1 -17757.59,E2 -17757.59} C_VEL
LIN {X 0,Y 289.54,Z 351.194,A -85,B 0,C 180,E1 -17758.155,E2 -17758.155} C_VEL
LIN {X 0,Y 291.89,Z 305.866,A -85,B 0,C 180,E1 -17759.532,E2 -17759.532} C_VEL
LIN {X 0,Y 289.986,Z 286.393,A -85,B 0,C 180,E1 -17760.593,E2 -17760.593} C_VEL
LIN {X 0,Y 287.297,Z 268.431,A -85,B 0,C 180,E1 -17761.781,E2 -17761.781} C_VEL
LIN {X 0,Y 285.976,Z 262.156,A -85,B 0,C 180,E1 -17762.28,E2 -17762.28} C_VEL
LIN {X 0,Y 281.673,Z 252.806,A -85,B 0,C 180,E1 -17763.489,E2 -17763.489} C_VEL
LIN {X 0,Y 278.875,Z 247.245,A -85,B 0,C 180,E1 -17764.301,E2 -17764.301} C_VEL
LIN {X 0,Y 276.929,Z 243.169,A -85,B 0,C 180,E1 -17764.933,E2 -17764.933} C_VEL
LIN {X 0,Y 274.957,Z 235.628,A -85,B 0,C 180,E1 -17767.839,E2 -17767.839} C_VEL
LIN {X 0,Y 272.272,Z 227.178,A -85,B 0,C 180,E1 -17771.534,E2 -17771.534} C_VEL
LIN {X 0,Y 270.152,Z 220.828,A -85,B 0,C 180,E1 -17774.75,E2 -17774.75} C_VEL
LIN {X 0,Y 270.145,Z 220.833,A -85,B 0,C 180,E1 -17778.977,E2 -17778.977} C_VEL
LIN {X 0,Y 270.207,Z 220.827,A -85,B 0,C 180,E1 -17781.374,E2 -17781.374} C_VEL
LIN {X 0,Y 270.198,Z 220.823,A -85,B 0,C 180,E1 -17785.094,E2 -17785.094} C_VEL
LIN {X 0,Y 270.184,Z 220.83,A -85,B 0,C 180,E1 -17789.136,E2 -17789.136} C_VEL
LIN {X 0,Y 270.223,Z 220.825,A -85,B 0,C 180,E1 -17792.162,E2 -17792.162} C_VEL
LIN {X 0,Y 270.229,Z 220.822,A -85,B 0,C 180,E1 -17795.541,E2 -17795.541} C_VEL
LIN {X 0,Y 270.263,Z 220.816,A -85,B 0,C 180,E1 -17800.241,E2 -17800.241} C_VEL
LIN {X 0,Y 270.373,Z 220.801,A -85,B 0,C 180,E1 -17804.934,E2 -17804.934} C_VEL
LIN {X 0,Y 270.413,Z 220.8,A -85,B 0,C 180,E1 -17809.518,E2 -17809.518} C_VEL
LIN {X 0,Y 270.599,Z 220.779,A -85,B 0,C 180,E1 -17812.538,E2 -17812.538} C_VEL
LIN {X 0,Y 270.786,Z 220.752,A -85,B 0,C 180,E1 -17818.513,E2 -17818.513} C_VEL
LIN {X 0,Y 270.742,Z 220.764,A -85,B 0,C 180,E1 -17821.813,E2 -17821.813} C_VEL
LIN {X 0,Y 271.607,Z 223.472,A -85,B 0,C 180,E1 -17822.178,E2 -17822.178} C_VEL
LIN {X 0,Y 273.813,Z 226.165,A -85,B 0,C 180,E1 -17822.85,E2 -17822.85} C_VEL
LIN {X 0,Y 275.648,Z 229.34,A -85,B 0,C 180,E1 -17823.425,E2 -17823.425} C_VEL
LIN {X 0,Y 277.177,Z 231.393,A -85,B 0,C 180,E1 -17823.861,E2 -17823.861} C_VEL
LIN {X 0,Y 282.411,Z 239.198,A -85,B 0,C 180,E1 -17825.319,E2 -17825.319} C_VEL
LIN {X 0,Y 289.253,Z 251.214,A -85,B 0,C 180,E1 -17827.109,E2 -17827.109} C_VEL
LIN {X 0,Y 293.976,Z 260.578,A -85,B 0,C 180,E1 -17828.293,E2 -17828.293} C_VEL
LIN {X 0,Y 290.5,Z 324.085,A -85,B 0,C 180,E1 -17830.256,E2 -17830.256} C_VEL
LIN {X 0,Y 289.466,Z 337.053,A -85,B 0,C 180,E1 -17830.934,E2 -17830.934} C_VEL
LIN {X 0,Y 287.954,Z 350.06,A -85,B 0,C 180,E1 -17831.904,E2 -17831.904} C_VEL
LIN {X 0,Y 285.98,Z 362.369,A -85,B 0,C 180,E1 -17833.139,E2 -17833.139} C_VEL
LIN {X 0,Y 283.856,Z 373.725,A -85,B 0,C 180,E1 -17834.614,E2 -17834.614} C_VEL
LIN {X 0,Y 281.448,Z 384.126,A -85,B 0,C 180,E1 -17836.315,E2 -17836.315} C_VEL
LIN {X 0,Y 279.055,Z 393.908,A -85,B 0,C 180,E1 -17838.349,E2 -17838.349} C_VEL
LIN {X 0,Y 276.81,Z 401.853,A -85,B 0,C 180,E1 -17840.436,E2 -17840.436} C_VEL
LIN {X 0,Y 274.591,Z 409.111,A -85,B 0,C 180,E1 -17842.869,E2 -17842.869} C_VEL
LIN {X 0,Y 273.084,Z 413.855,A -85,B 0,C 180,E1 -17844.916,E2 -17844.916} C_VEL
LIN {X 0,Y 271.36,Z 418.83,A -85,B 0,C 180,E1 -17847.787,E2 -17847.787} C_VEL
LIN {X 0,Y 270.494,Z 421.047,A -85,B 0,C 180,E1 -17849.581,E2 -17849.581} C_VEL
LIN {X 0,Y 269.803,Z 422.619,A -85,B 0,C 180,E1 -17851.397,E2 -17851.397} C_VEL
LIN {X 0,Y 269.214,Z 423.655,A -85,B 0,C 180,E1 -17853.345,E2 -17853.345} C_VEL
LIN {X 0,Y 268.726,Z 423.935,A -85,B 0,C 180,E1 -17855.832,E2 -17855.832} C_VEL
LIN {X 0,Y 268.514,Z 423.128,A -85,B 0,C 180,E1 -17858.261,E2 -17858.261} C_VEL
LIN {X 0,Y 268.585,Z 421.065,A -85,B 0,C 180,E1 -17860.857,E2 -17860.857} C_VEL
LIN {X 0,Y 268.909,Z 418.461,A -85,B 0,C 180,E1 -17862.964,E2 -17862.964} C_VEL
LIN {X 0,Y 269.323,Z 414.684,A -85,B 0,C 180,E1 -17865.206,E2 -17865.206} C_VEL
LIN {X 0,Y 269.908,Z 409.894,A -85,B 0,C 180,E1 -17867.391,E2 -17867.391} C_VEL
LIN {X 0,Y 270.789,Z 403.12,A -85,B 0,C 180,E1 -17869.81,E2 -17869.81} C_VEL
LIN {X 0,Y 271.922,Z 394.791,A -85,B 0,C 180,E1 -17872.159,E2 -17872.159} C_VEL
LIN {X 0,Y 273.213,Z 385.259,A -85,B 0,C 180,E1 -17874.283,E2 -17874.283} C_VEL
LIN {X 0,Y 274.585,Z 374.957,A -85,B 0,C 180,E1 -17876.129,E2 -17876.129} C_VEL
LIN {X 0,Y 275.753,Z 364.419,A -85,B 0,C 180,E1 -17877.642,E2 -17877.642} C_VEL
LIN {X 0,Y 277.104,Z 351.66,A -85,B 0,C 180,E1 -17879.081,E2 -17879.081} C_VEL
LIN {X 0,Y 278.134,Z 338.852,A -85,B 0,C 180,E1 -17880.168,E2 -17880.168} C_VEL
LIN {X 0,Y 278.837,Z 325.198,A -85,B 0,C 180,E1 -17881.001,E2 -17881.001} C_VEL
LIN {X 0,Y 279.374,Z 311.462,A -85,B 0,C 180,E1 -17881.518,E2 -17881.518} C_VEL
LIN {X 0,Y 281.372,Z 249.33,A -85,B 0,C 180,E1 -17883.354,E2 -17883.354} C_VEL
LIN {X 0,Y 270.996,Z 223.118,A -85,B 0,C 180,E1 -17885.005,E2 -17885.005} C_VEL
LIN {X 0,Y 270.263,Z 220.823,A -85,B 0,C 180,E1 -17885.183,E2 -17885.183} C_VEL
LIN {X 0,Y 270.262,Z 220.819,A -85,B 0,C 180,E1 -17890.242,E2 -17890.242} C_VEL
LIN {X 0,Y 270.378,Z 220.807,A -85,B 0,C 180,E1 -17894.934,E2 -17894.934} C_VEL
LIN {X 0,Y 270.411,Z 220.8,A -85,B 0,C 180,E1 -17899.518,E2 -17899.518} C_VEL
LIN {X 0,Y 270.566,Z 220.784,A -85,B 0,C 180,E1 -17902.538,E2 -17902.538} C_VEL
LIN {X 0,Y 270.785,Z 220.757,A -85,B 0,C 180,E1 -17908.513,E2 -17908.513} C_VEL
LIN {X 0,Y 270.783,Z 220.752,A -85,B 0,C 180,E1 -17911.488,E2 -17911.488} C_VEL
LIN {X 0,Y 270.572,Z 220.779,A -85,B 0,C 180,E1 -17917.463,E2 -17917.463} C_VEL
LIN {X 0,Y 270.414,Z 220.801,A -85,B 0,C 180,E1 -17920.483,E2 -17920.483} C_VEL
LIN {X 0,Y 270.405,Z 220.8,A -85,B 0,C 180,E1 -17925.065,E2 -17925.065} C_VEL
LIN {X 0,Y 270.302,Z 220.813,A -85,B 0,C 180,E1 -17929.756,E2 -17929.756} C_VEL
LIN {X 0,Y 270.228,Z 220.82,A -85,B 0,C 180,E1 -17934.591,E2 -17934.591} C_VEL
LIN {X 0,Y 270.205,Z 220.829,A -85,B 0,C 180,E1 -17937.917,E2 -17937.917} C_VEL
LIN {X 0,Y 270.175,Z 220.83,A -85,B 0,C 180,E1 -17941.35,E2 -17941.35} C_VEL
LIN {X 0,Y 270.199,Z 220.821,A -85,B 0,C 180,E1 -17944.906,E2 -17944.906} C_VEL
LIN {X 0,Y 270.199,Z 220.815,A -85,B 0,C 180,E1 -17948.711,E2 -17948.711} C_VEL
LIN {X 0,Y 270.162,Z 220.83,A -85,B 0,C 180,E1 -17953.248,E2 -17953.248} C_VEL
LIN {X 0,Y 270.157,Z 220.835,A -85,B 0,C 180,E1 -17957.439,E2 -17957.439} C_VEL
LIN {X 0,Y 270.209,Z 220.825,A -85,B 0,C 180,E1 -17961.375,E2 -17961.375} C_VEL
LIN {X 0,Y 270.203,Z 220.826,A -85,B 0,C 180,E1 -17965.095,E2 -17965.095} C_VEL
LIN {X 0,Y 270.186,Z 220.831,A -85,B 0,C 180,E1 -17969.137,E2 -17969.137} C_VEL
LIN {X 0,Y 270.225,Z 220.821,A -85,B 0,C 180,E1 -17972.163,E2 -17972.163} C_VEL
LIN {X 0,Y 270.23,Z 220.82,A -85,B 0,C 180,E1 -17975.543,E2 -17975.543} C_VEL
LIN {X 0,Y 270.264,Z 220.818,A -85,B 0,C 180,E1 -17980.242,E2 -17980.242} C_VEL
LIN {X 0,Y 270.38,Z 220.802,A -85,B 0,C 180,E1 -17984.934,E2 -17984.934} C_VEL
LIN {X 0,Y 270.413,Z 220.787,A -85,B 0,C 180,E1 -17989.518,E2 -17989.518} C_VEL
LIN {X 0,Y 270.566,Z 220.775,A -85,B 0,C 180,E1 -17992.538,E2 -17992.538} C_VEL
LIN {X 0,Y 270.669,Z 220.766,A -85,B 0,C 180,E1 -17997.697,E2 -17997.697} C_VEL
LIN {X 0,Y 270.417,Z 220.802,A -85,B 0,C 180,E1 -17998.528,E2 -17998.528} C_VEL
LIN {X 0,Y 269.094,Z 220.965,A -85,B 0,C 180,E1 -17999.755,E2 -17999.755} C_VEL
LIN {X 0,Y 264.622,Z 221.521,A -85,B 0,C 180,E1 -18002.607,E2 -18002.607} C_VEL
LIN {X 0,Y 263.478,Z 221.663,A -85,B 0,C 180,E1 -18003.885,E2 -18003.885} C_VEL
LIN {X 0,Y 263.364,Z 221.673,A -85,B 0,C 180,E1 -18004.319,E2 -18004.319} C_VEL
LIN {X 0,Y 263.529,Z 221.65,A -85,B 0,C 180,E1 -18007.663,E2 -18007.663} C_VEL
LIN {X 0,Y 263.353,Z 221.676,A -85,B 0,C 180,E1 -18010.767,E2 -18010.767} C_VEL
LIN {X 0,Y 263.302,Z 221.687,A -85,B 0,C 180,E1 -18015.481,E2 -18015.481} C_VEL
LIN {X 0,Y 263.24,Z 221.689,A -85,B 0,C 180,E1 -18020.309,E2 -18020.309} C_VEL
LIN {X 0,Y 263.13,Z 221.708,A -85,B 0,C 180,E1 -18025.3,E2 -18025.3} C_VEL
LIN {X 0,Y 263.135,Z 221.705,A -85,B 0,C 180,E1 -18028.735,E2 -18028.735} C_VEL
LIN {X 0,Y 263.131,Z 221.706,A -85,B 0,C 180,E1 -18032.289,E2 -18032.289} C_VEL
LIN {X 0,Y 263.178,Z 221.7,A -85,B 0,C 180,E1 -18036.761,E2 -18036.761} C_VEL
LIN {X 0,Y 263.093,Z 221.714,A -85,B 0,C 180,E1 -18039.875,E2 -18039.875} C_VEL
LIN {X 0,Y 263.078,Z 221.714,A -85,B 0,C 180,E1 -18043.994,E2 -18043.994} C_VEL
LIN {X 0,Y 263.082,Z 221.713,A -85,B 0,C 180,E1 -18048.417,E2 -18048.417} C_VEL
LIN {X 0,Y 263.162,Z 221.704,A -85,B 0,C 180,E1 -18052.103,E2 -18052.103} C_VEL
LIN {X 0,Y 263.219,Z 221.789,A -85,B 0,C 180,E1 -18053.635,E2 -18053.635} C_VEL
LIN {X 0,Y 265.985,Z 234.637,A -85,B 0,C 180,E1 -18057.728,E2 -18057.728} C_VEL
LIN {X 0,Y 268.145,Z 245.377,A -85,B 0,C 180,E1 -18060.995,E2 -18060.995} C_VEL
LIN {X 0,Y 267.738,Z 250.124,A -85,B 0,C 180,E1 -18062.321,E2 -18062.321} C_VEL
LIN {X 0,Y 273.478,Z 303.927,A -85,B 0,C 180,E1 -18064.559,E2 -18064.559} C_VEL
LIN {X 0,Y 271.648,Z 359.863,A -85,B 0,C 180,E1 -18066.307,E2 -18066.307} C_VEL
LIN {X 0,Y 270.707,Z 373.66,A -85,B 0,C 180,E1 -18067.03,E2 -18067.03} C_VEL
LIN {X 0,Y 269.492,Z 386.195,A -85,B 0,C 180,E1 -18067.983,E2 -18067.983} C_VEL
LIN {X 0,Y 267.946,Z 398.617,A -85,B 0,C 180,E1 -18069.262,E2 -18069.262} C_VEL
LIN {X 0,Y 266.494,Z 409.848,A -85,B 0,C 180,E1 -18070.752,E2 -18070.752} C_VEL
LIN {X 0,Y 265.126,Z 419.377,A -85,B 0,C 180,E1 -18072.33,E2 -18072.33} C_VEL
LIN {X 0,Y 263.889,Z 428.564,A -85,B 0,C 180,E1 -18074.211,E2 -18074.211} C_VEL
LIN {X 0,Y 262.819,Z 437.466,A -85,B 0,C 180,E1 -18076.468,E2 -18076.468} C_VEL
LIN {X 0,Y 261.948,Z 444.743,A -85,B 0,C 180,E1 -18078.783,E2 -18078.783} C_VEL
LIN {X 0,Y 261.631,Z 449.661,A -85,B 0,C 180,E1 -18080.725,E2 -18080.725} C_VEL
LIN {X 0,Y 261.509,Z 454.373,A -85,B 0,C 180,E1 -18083.053,E2 -18083.053} C_VEL
LIN {X 0,Y 261.527,Z 457.887,A -85,B 0,C 180,E1 -18085.375,E2 -18085.375} C_VEL
LIN {X 0,Y 261.51,Z 459.591,A -85,B 0,C 180,E1 -18086.918,E2 -18086.918} C_VEL
LIN {X 0,Y 261.714,Z 460.868,A -85,B 0,C 180,E1 -18088.461,E2 -18088.461} C_VEL
LIN {X 0,Y 261.811,Z 461.709,A -85,B 0,C 180,E1 -18090,E2 -18090} C_VEL
LIN {X 0,Y 261.601,Z 462.084,A -85,B 0,C 180,E1 -18091.539,E2 -18091.539} C_VEL
LIN {X 0,Y 261.389,Z 462.008,A -85,B 0,C 180,E1 -18093.082,E2 -18093.082} C_VEL
LIN {X 0,Y 261.21,Z 461.134,A -85,B 0,C 180,E1 -18095.432,E2 -18095.432} C_VEL
LIN {X 0,Y 261.316,Z 459.372,A -85,B 0,C 180,E1 -18097.728,E2 -18097.728} C_VEL
LIN {X 0,Y 261.656,Z 456.626,A -85,B 0,C 180,E1 -18100.054,E2 -18100.054} C_VEL
LIN {X 0,Y 262.345,Z 452.869,A -85,B 0,C 180,E1 -18102.375,E2 -18102.375} C_VEL
LIN {X 0,Y 263.67,Z 448.055,A -85,B 0,C 180,E1 -18104.668,E2 -18104.668} C_VEL
LIN {X 0,Y 265.558,Z 440.924,A -85,B 0,C 180,E1 -18107.302,E2 -18107.302} C_VEL
LIN {X 0,Y 267.605,Z 433.172,A -85,B 0,C 180,E1 -18109.563,E2 -18109.563} C_VEL
LIN {X 0,Y 269.817,Z 425.396,A -85,B 0,C 180,E1 -18111.386,E2 -18111.386} C_VEL
LIN {X 0,Y 272.398,Z 416.061,A -85,B 0,C 180,E1 -18113.169,E2 -18113.169} C_VEL
LIN {X 0,Y 275.177,Z 404.594,A -85,B 0,C 180,E1 -18114.923,E2 -18114.923} C_VEL
LIN {X 0,Y 277.794,Z 393.181,A -85,B 0,C 180,E1 -18116.278,E2 -18116.278} C_VEL
LIN {X 0,Y 280.254,Z 380.385,A -85,B 0,C 180,E1 -18117.438,E2 -18117.438} C_VEL
LIN {X 0,Y 282.314,Z 366.904,A -85,B 0,C 180,E1 -18118.325,E2 -18118.325} C_VEL
LIN {X 0,Y 283.66,Z 354.184,A -85,B 0,C 180,E1 -18118.9,E2 -18118.9} C_VEL
LIN {X 0,Y 286.225,Z 306.32,A -85,B 0,C 180,E1 -18120.406,E2 -18120.406} C_VEL
LIN {X 0,Y 284.576,Z 288.267,A -85,B 0,C 180,E1 -18121.43,E2 -18121.43} C_VEL
LIN {X 0,Y 281.986,Z 270.015,A -85,B 0,C 180,E1 -18122.68,E2 -18122.68} C_VEL
LIN {X 0,Y 280.981,Z 265.557,A -85,B 0,C 180,E1 -18123.06,E2 -18123.06} C_VEL
LIN {X 0,Y 276.729,Z 256.165,A -85,B 0,C 180,E1 -18124.338,E2 -18124.338} C_VEL
LIN {X 0,Y 274.135,Z 250.949,A -85,B 0,C 180,E1 -18125.139,E2 -18125.139} C_VEL
LIN {X 0,Y 271.88,Z 246.701,A -85,B 0,C 180,E1 -18125.852,E2 -18125.852} C_VEL
LIN {X 0,Y 269.581,Z 242.074,A -85,B 0,C 180,E1 -18126.691,E2 -18126.691} C_VEL
LIN {X 0,Y 267.608,Z 235.292,A -85,B 0,C 180,E1 -18129.564,E2 -18129.564} C_VEL
LIN {X 0,Y 265.764,Z 229.623,A -85,B 0,C 180,E1 -18132.23,E2 -18132.23} C_VEL
LIN {X 0,Y 263.106,Z 221.709,A -85,B 0,C 180,E1 -18136.536,E2 -18136.536} C_VEL
LIN {X 0,Y 263.112,Z 221.709,A -85,B 0,C 180,E1 -18140.77,E2 -18140.77} C_VEL
LIN {X 0,Y 263.159,Z 221.704,A -85,B 0,C 180,E1 -18144.017,E2 -18144.017} C_VEL
LIN {X 0,Y 263.128,Z 221.702,A -85,B 0,C 180,E1 -18147.711,E2 -18147.711} C_VEL
LIN {X 0,Y 263.151,Z 221.705,A -85,B 0,C 180,E1 -18151.803,E2 -18151.803} C_VEL
LIN {X 0,Y 263.191,Z 221.702,A -85,B 0,C 180,E1 -18155.217,E2 -18155.217} C_VEL
LIN {X 0,Y 263.239,Z 221.688,A -85,B 0,C 180,E1 -18159.691,E2 -18159.691} C_VEL
LIN {X 0,Y 263.314,Z 221.683,A -85,B 0,C 180,E1 -18164.52,E2 -18164.52} C_VEL
LIN {X 0,Y 263.355,Z 221.677,A -85,B 0,C 180,E1 -18169.233,E2 -18169.233} C_VEL
LIN {X 0,Y 263.558,Z 221.656,A -85,B 0,C 180,E1 -18172.338,E2 -18172.338} C_VEL
LIN {X 0,Y 263.75,Z 221.628,A -85,B 0,C 180,E1 -18178.473,E2 -18178.473} C_VEL
LIN {X 0,Y 263.827,Z 221.811,A -85,B 0,C 180,E1 -18180.048,E2 -18180.048} C_VEL
LIN {X 0,Y 264.672,Z 224.299,A -85,B 0,C 180,E1 -18180.428,E2 -18180.428} C_VEL
LIN {X 0,Y 266.708,Z 226.541,A -85,B 0,C 180,E1 -18181.101,E2 -18181.101} C_VEL
LIN {X 0,Y 267.847,Z 228.574,A -85,B 0,C 180,E1 -18181.503,E2 -18181.503} C_VEL
LIN {X 0,Y 270.115,Z 231.677,A -85,B 0,C 180,E1 -18182.237,E2 -18182.237} C_VEL
LIN {X 0,Y 272.603,Z 235.527,A -85,B 0,C 180,E1 -18183.038,E2 -18183.038} C_VEL
LIN {X 0,Y 278.445,Z 244.419,A -85,B 0,C 180,E1 -18184.741,E2 -18184.741} C_VEL
LIN {X 0,Y 283.985,Z 254.299,A -85,B 0,C 180,E1 -18186.281,E2 -18186.281} C_VEL
LIN {X 0,Y 288.415,Z 263.102,A -85,B 0,C 180,E1 -18187.457,E2 -18187.457} C_VEL
LIN {X 0,Y 284.842,Z 324.597,A -85,B 0,C 180,E1 -18189.408,E2 -18189.408} C_VEL
LIN {X 0,Y 283.77,Z 337.541,A -85,B 0,C 180,E1 -18190.096,E2 -18190.096} C_VEL
LIN {X 0,Y 282.237,Z 350.102,A -85,B 0,C 180,E1 -18191.036,E2 -18191.036} C_VEL
LIN {X 0,Y 280.39,Z 361.459,A -85,B 0,C 180,E1 -18192.168,E2 -18192.168} C_VEL
LIN {X 0,Y 278.327,Z 371.998,A -85,B 0,C 180,E1 -18193.507,E2 -18193.507} C_VEL
LIN {X 0,Y 276.044,Z 381.987,A -85,B 0,C 180,E1 -18195.089,E2 -18195.089} C_VEL
LIN {X 0,Y 273.939,Z 390.133,A -85,B 0,C 180,E1 -18196.676,E2 -18196.676} C_VEL
LIN {X 0,Y 271.329,Z 399.29,A -85,B 0,C 180,E1 -18198.891,E2 -18198.891} C_VEL
LIN {X 0,Y 269.357,Z 405.656,A -85,B 0,C 180,E1 -18200.814,E2 -18200.814} C_VEL
LIN {X 0,Y 267.237,Z 412.001,A -85,B 0,C 180,E1 -18203.234,E2 -18203.234} C_VEL
LIN {X 0,Y 265.439,Z 417.129,A -85,B 0,C 180,E1 -18205.815,E2 -18205.815} C_VEL
LIN {X 0,Y 263.858,Z 421.056,A -85,B 0,C 180,E1 -18208.649,E2 -18208.649} C_VEL
LIN {X 0,Y 262.813,Z 423.267,A -85,B 0,C 180,E1 -18211.161,E2 -18211.161} C_VEL
LIN {X 0,Y 261.93,Z 424.49,A -85,B 0,C 180,E1 -18214.296,E2 -18214.296} C_VEL
LIN {X 0,Y 261.577,Z 424.354,A -85,B 0,C 180,E1 -18216.29,E2 -18216.29} C_VEL
LIN {X 0,Y 261.428,Z 423.246,A -85,B 0,C 180,E1 -18218.776,E2 -18218.776} C_VEL
LIN {X 0,Y 261.535,Z 421.125,A -85,B 0,C 180,E1 -18221.2,E2 -18221.2} C_VEL
LIN {X 0,Y 262.047,Z 416.963,A -85,B 0,C 180,E1 -18224.212,E2 -18224.212} C_VEL
LIN {X 0,Y 262.532,Z 413.039,A -85,B 0,C 180,E1 -18226.285,E2 -18226.285} C_VEL
LIN {X 0,Y 263.32,Z 406.738,A -85,B 0,C 180,E1 -18228.867,E2 -18228.867} C_VEL
LIN {X 0,Y 264.203,Z 400.188,A -85,B 0,C 180,E1 -18230.998,E2 -18230.998} C_VEL
LIN {X 0,Y 265.343,Z 392.382,A -85,B 0,C 180,E1 -18233.063,E2 -18233.063} C_VEL
LIN {X 0,Y 266.685,Z 382.396,A -85,B 0,C 180,E1 -18235.187,E2 -18235.187} C_VEL
LIN {X 0,Y 268.079,Z 371.588,A -85,B 0,C 180,E1 -18237.026,E2 -18237.026} C_VEL
LIN {X 0,Y 269.366,Z 360.318,A -85,B 0,C 180,E1 -18238.546,E2 -18238.546} C_VEL
LIN {X 0,Y 270.691,Z 347.282,A -85,B 0,C 180,E1 -18239.907,E2 -18239.907} C_VEL
LIN {X 0,Y 271.698,Z 334.242,A -85,B 0,C 180,E1 -18240.911,E2 -18240.911} C_VEL
LIN {X 0,Y 272.255,Z 321.888,A -85,B 0,C 180,E1 -18241.585,E2 -18241.585} C_VEL
LIN {X 0,Y 273.291,Z 291.932,A -85,B 0,C 180,E1 -18242.55,E2 -18242.55} C_VEL
LIN {X 0,Y 274.738,Z 251.104,A -85,B 0,C 180,E1 -18243.785,E2 -18243.785} C_VEL
LIN {X 0,Y 264.158,Z 224.404,A -85,B 0,C 180,E1 -18245.514,E2 -18245.514} C_VEL
LIN {X 0,Y 263.215,Z 221.698,A -85,B 0,C 180,E1 -18245.713,E2 -18245.713} C_VEL
LIN {X 0,Y 263.239,Z 221.694,A -85,B 0,C 180,E1 -18249.692,E2 -18249.692} C_VEL
LIN {X 0,Y 263.324,Z 221.685,A -85,B 0,C 180,E1 -18254.521,E2 -18254.521} C_VEL
LIN {X 0,Y 263.35,Z 221.681,A -85,B 0,C 180,E1 -18259.234,E2 -18259.234} C_VEL
LIN {X 0,Y 263.529,Z 221.659,A -85,B 0,C 180,E1 -18262.338,E2 -18262.338} C_VEL
LIN {X 0,Y 263.749,Z 221.633,A -85,B 0,C 180,E1 -18268.474,E2 -18268.474} C_VEL
LIN {X 0,Y 263.747,Z 221.629,A -85,B 0,C 180,E1 -18271.527,E2 -18271.527} C_VEL
LIN {X 0,Y 263.534,Z 221.656,A -85,B 0,C 180,E1 -18277.663,E2 -18277.663} C_VEL
LIN {X 0,Y 263.356,Z 221.679,A -85,B 0,C 180,E1 -18280.767,E2 -18280.767} C_VEL
LIN {X 0,Y 263.353,Z 221.679,A -85,B 0,C 180,E1 -18285.478,E2 -18285.478} C_VEL
LIN {X 0,Y 263.264,Z 221.686,A -85,B 0,C 180,E1 -18290.307,E2 -18290.307} C_VEL
LIN {X 0,Y 263.172,Z 221.699,A -85,B 0,C 180,E1 -18295.296,E2 -18295.296} C_VEL
LIN {X 0,Y 263.138,Z 221.705,A -85,B 0,C 180,E1 -18298.735,E2 -18298.735} C_VEL
LIN {X 0,Y 263.13,Z 221.705,A -85,B 0,C 180,E1 -18302.289,E2 -18302.289} C_VEL
LIN {X 0,Y 263.177,Z 221.69,A -85,B 0,C 180,E1 -18306.762,E2 -18306.762} C_VEL
LIN {X 0,Y 263.104,Z 221.704,A -85,B 0,C 180,E1 -18309.873,E2 -18309.873} C_VEL
LIN {X 0,Y 263.104,Z 221.709,A -85,B 0,C 180,E1 -18313.989,E2 -18313.989} C_VEL
LIN {X 0,Y 263.111,Z 221.708,A -85,B 0,C 180,E1 -18318.411,E2 -18318.411} C_VEL
LIN {X 0,Y 263.16,Z 221.699,A -85,B 0,C 180,E1 -18322.103,E2 -18322.103} C_VEL
LIN {X 0,Y 263.153,Z 221.703,A -85,B 0,C 180,E1 -18325.886,E2 -18325.886} C_VEL
LIN {X 0,Y 263.128,Z 221.708,A -85,B 0,C 180,E1 -18329.504,E2 -18329.504} C_VEL
LIN {X 0,Y 263.144,Z 221.705,A -85,B 0,C 180,E1 -18332.997,E2 -18332.997} C_VEL
LIN {X 0,Y 263.148,Z 221.702,A -85,B 0,C 180,E1 -18336.384,E2 -18336.384} C_VEL
LIN {X 0,Y 263.241,Z 221.692,A -85,B 0,C 180,E1 -18339.692,E2 -18339.692} C_VEL
LIN {X 0,Y 263.326,Z 221.682,A -85,B 0,C 180,E1 -18344.521,E2 -18344.521} C_VEL
LIN {X 0,Y 263.352,Z 221.666,A -85,B 0,C 180,E1 -18349.234,E2 -18349.234} C_VEL
LIN {X 0,Y 263.529,Z 221.648,A -85,B 0,C 180,E1 -18352.337,E2 -18352.337} C_VEL
LIN {X 0,Y 263.744,Z 221.634,A -85,B 0,C 180,E1 -18358.473,E2 -18358.473} C_VEL
LIN {X 0,Y 263.741,Z 221.63,A -85,B 0,C 180,E1 -18361.527,E2 -18361.527} C_VEL
LIN {X 0,Y 263.364,Z 221.673,A -85,B 0,C 180,E1 -18364.319,E2 -18364.319} C_VEL
LIN {X 0,Y 262.656,Z 221.767,A -85,B 0,C 180,E1 -18365.596,E2 -18365.596} C_VEL
LIN {X 0,Y 259.847,Z 222.122,A -85,B 0,C 180,E1 -18367.681,E2 -18367.681} C_VEL
LIN {X 0,Y 256.646,Z 222.515,A -85,B 0,C 180,E1 -18370.245,E2 -18370.245} C_VEL
LIN {X 0,Y 256.287,Z 222.555,A -85,B 0,C 180,E1 -18371.131,E2 -18371.131} C_VEL
LIN {X 0,Y 256.24,Z 222.569,A -85,B 0,C 180,E1 -18375.919,E2 -18375.919} C_VEL
LIN {X 0,Y 256.147,Z 222.571,A -85,B 0,C 180,E1 -18380.897,E2 -18380.897} C_VEL
LIN {X 0,Y 256.089,Z 222.585,A -85,B 0,C 180,E1 -18385.089,E2 -18385.089} C_VEL
LIN {X 0,Y 256.092,Z 222.583,A -85,B 0,C 180,E1 -18388.575,E2 -18388.575} C_VEL
LIN {X 0,Y 256.077,Z 222.587,A -85,B 0,C 180,E1 -18391.701,E2 -18391.701} C_VEL
LIN {X 0,Y 256.082,Z 222.586,A -85,B 0,C 180,E1 -18395.193,E2 -18395.193} C_VEL
LIN {X 0,Y 256.113,Z 222.583,A -85,B 0,C 180,E1 -18397.269,E2 -18397.269} C_VEL
LIN {X 0,Y 256.042,Z 222.594,A -85,B 0,C 180,E1 -18401.206,E2 -18401.206} C_VEL
LIN {X 0,Y 256.02,Z 222.595,A -85,B 0,C 180,E1 -18405.539,E2 -18405.539} C_VEL
LIN {X 0,Y 256.021,Z 222.594,A -85,B 0,C 180,E1 -18408.789,E2 -18408.789} C_VEL
LIN {X 0,Y 256.188,Z 222.747,A -85,B 0,C 180,E1 -18413.245,E2 -18413.245} C_VEL
LIN {X 0,Y 259.023,Z 235.903,A -85,B 0,C 180,E1 -18417.555,E2 -18417.555} C_VEL
LIN {X 0,Y 261.033,Z 245.745,A -85,B 0,C 180,E1 -18420.628,E2 -18420.628} C_VEL
LIN {X 0,Y 261.011,Z 249.136,A -85,B 0,C 180,E1 -18421.621,E2 -18421.621} C_VEL
LIN {X 0,Y 260.933,Z 249.623,A -85,B 0,C 180,E1 -18421.758,E2 -18421.758} C_VEL
LIN {X 0,Y 266.708,Z 305.455,A -85,B 0,C 180,E1 -18424.141,E2 -18424.141} C_VEL
LIN {X 0,Y 264.812,Z 360.264,A -85,B 0,C 180,E1 -18425.917,E2 -18425.917} C_VEL
LIN {X 0,Y 263.825,Z 373.741,A -85,B 0,C 180,E1 -18426.655,E2 -18426.655} C_VEL
LIN {X 0,Y 262.65,Z 385.581,A -85,B 0,C 180,E1 -18427.585,E2 -18427.585} C_VEL
LIN {X 0,Y 261.067,Z 398.008,A -85,B 0,C 180,E1 -18428.896,E2 -18428.896} C_VEL
LIN {X 0,Y 259.573,Z 409.246,A -85,B 0,C 180,E1 -18430.424,E2 -18430.424} C_VEL
LIN {X 0,Y 258.075,Z 419.388,A -85,B 0,C 180,E1 -18432.159,E2 -18432.159} C_VEL
LIN {X 0,Y 256.821,Z 428.6,A -85,B 0,C 180,E1 -18434.118,E2 -18434.118} C_VEL
LIN {X 0,Y 255.703,Z 437.587,A -85,B 0,C 180,E1 -18436.489,E2 -18436.489} C_VEL
LIN {X 0,Y 254.853,Z 444.702,A -85,B 0,C 180,E1 -18438.869,E2 -18438.869} C_VEL
LIN {X 0,Y 254.5,Z 450.377,A -85,B 0,C 180,E1 -18441.264,E2 -18441.264} C_VEL
LIN {X 0,Y 254.46,Z 455.13,A -85,B 0,C 180,E1 -18443.878,E2 -18443.878} C_VEL
LIN {X 0,Y 254.47,Z 457.069,A -85,B 0,C 180,E1 -18445.247,E2 -18445.247} C_VEL
LIN {X 0,Y 254.434,Z 458.861,A -85,B 0,C 180,E1 -18446.833,E2 -18446.833} C_VEL
LIN {X 0,Y 254.624,Z 460.182,A -85,B 0,C 180,E1 -18448.418,E2 -18448.418} C_VEL
LIN {X 0,Y 254.756,Z 461.069,A -85,B 0,C 180,E1 -18450,E2 -18450} C_VEL
LIN {X 0,Y 254.51,Z 461.503,A -85,B 0,C 180,E1 -18451.582,E2 -18451.582} C_VEL
LIN {X 0,Y 254.31,Z 461.491,A -85,B 0,C 180,E1 -18453.168,E2 -18453.168} C_VEL
LIN {X 0,Y 254.124,Z 460.797,A -85,B 0,C 180,E1 -18455.368,E2 -18455.368} C_VEL
LIN {X 0,Y 254.245,Z 458.99,A -85,B 0,C 180,E1 -18457.944,E2 -18457.944} C_VEL
LIN {X 0,Y 254.634,Z 456.328,A -85,B 0,C 180,E1 -18460.335,E2 -18460.335} C_VEL
LIN {X 0,Y 255.379,Z 452.679,A -85,B 0,C 180,E1 -18462.718,E2 -18462.718} C_VEL
LIN {X 0,Y 256.785,Z 447.966,A -85,B 0,C 180,E1 -18465.07,E2 -18465.07} C_VEL
LIN {X 0,Y 258.469,Z 442.061,A -85,B 0,C 180,E1 -18467.403,E2 -18467.403} C_VEL
LIN {X 0,Y 260.512,Z 434.773,A -85,B 0,C 180,E1 -18469.707,E2 -18469.707} C_VEL
LIN {X 0,Y 263.229,Z 425.805,A -85,B 0,C 180,E1 -18471.949,E2 -18471.949} C_VEL
LIN {X 0,Y 266.203,Z 415.724,A -85,B 0,C 180,E1 -18473.948,E2 -18473.948} C_VEL
LIN {X 0,Y 269.117,Z 404.337,A -85,B 0,C 180,E1 -18475.732,E2 -18475.732} C_VEL
LIN {X 0,Y 271.867,Z 392.982,A -85,B 0,C 180,E1 -18477.104,E2 -18477.104} C_VEL
LIN {X 0,Y 274.431,Z 380.335,A -85,B 0,C 180,E1 -18478.279,E2 -18478.279} C_VEL
LIN {X 0,Y 276.592,Z 366.955,A -85,B 0,C 180,E1 -18479.179,E2 -18479.179} C_VEL
LIN {X 0,Y 278.054,Z 353.988,A -85,B 0,C 180,E1 -18479.79,E2 -18479.79} C_VEL
LIN {X 0,Y 280.764,Z 307.552,A -85,B 0,C 180,E1 -18481.292,E2 -18481.292} C_VEL
LIN {X 0,Y 279.201,Z 289.43,A -85,B 0,C 180,E1 -18482.352,E2 -18482.352} C_VEL
LIN {X 0,Y 276.826,Z 272.228,A -85,B 0,C 180,E1 -18483.578,E2 -18483.578} C_VEL
LIN {X 0,Y 276.09,Z 268.91,A -85,B 0,C 180,E1 -18483.882,E2 -18483.882} C_VEL
LIN {X 0,Y 271.145,Z 257.815,A -85,B 0,C 180,E1 -18485.47,E2 -18485.47} C_VEL
LIN {X 0,Y 267.492,Z 250.841,A -85,B 0,C 180,E1 -18486.687,E2 -18486.687} C_VEL
LIN {X 0,Y 264.925,Z 246.131,A -85,B 0,C 180,E1 -18487.584,E2 -18487.584} C_VEL
LIN {X 0,Y 262.164,Z 241.087,A -85,B 0,C 180,E1 -18488.642,E2 -18488.642} C_VEL
LIN {X 0,Y 259.57,Z 232.814,A -85,B 0,C 180,E1 -18492.601,E2 -18492.601} C_VEL
LIN {X 0,Y 256.978,Z 225.254,A -85,B 0,C 180,E1 -18496.865,E2 -18496.865} C_VEL
LIN {X 0,Y 256.051,Z 222.591,A -85,B 0,C 180,E1 -18498.656,E2 -18498.656} C_VEL
LIN {X 0,Y 256.127,Z 222.577,A -85,B 0,C 180,E1 -18502.867,E2 -18502.867} C_VEL
LIN {X 0,Y 256.065,Z 222.587,A -85,B 0,C 180,E1 -18506.707,E2 -18506.707} C_VEL
LIN {X 0,Y 256.056,Z 222.583,A -85,B 0,C 180,E1 -18510.393,E2 -18510.393} C_VEL
LIN {X 0,Y 256.134,Z 222.581,A -85,B 0,C 180,E1 -18514.887,E2 -18514.887} C_VEL
LIN {X 0,Y 256.148,Z 222.572,A -85,B 0,C 180,E1 -18519.103,E2 -18519.103} C_VEL
LIN {X 0,Y 256.248,Z 222.566,A -85,B 0,C 180,E1 -18524.082,E2 -18524.082} C_VEL
LIN {X 0,Y 256.29,Z 222.558,A -85,B 0,C 180,E1 -18527.327,E2 -18527.327} C_VEL
LIN {X 0,Y 256.515,Z 222.532,A -85,B 0,C 180,E1 -18532.126,E2 -18532.126} C_VEL
LIN {X 0,Y 256.633,Z 222.517,A -85,B 0,C 180,E1 -18537.891,E2 -18537.891} C_VEL
LIN {X 0,Y 257.475,Z 225.004,A -85,B 0,C 180,E1 -18538.338,E2 -18538.338} C_VEL
LIN {X 0,Y 259.614,Z 227.397,A -85,B 0,C 180,E1 -18539.147,E2 -18539.147} C_VEL
LIN {X 0,Y 260.44,Z 228.093,A -85,B 0,C 180,E1 -18539.436,E2 -18539.436} C_VEL
LIN {X 0,Y 262.519,Z 231.518,A -85,B 0,C 180,E1 -18540.24,E2 -18540.24} C_VEL
LIN {X 0,Y 263.935,Z 233.323,A -85,B 0,C 180,E1 -18540.739,E2 -18540.739} C_VEL
LIN {X 0,Y 267.284,Z 238.539,A -85,B 0,C 180,E1 -18541.89,E2 -18541.89} C_VEL
LIN {X 0,Y 274.181,Z 249.023,A -85,B 0,C 180,E1 -18544.047,E2 -18544.047} C_VEL
LIN {X 0,Y 279.506,Z 258.766,A -85,B 0,C 180,E1 -18545.623,E2 -18545.623} C_VEL
LIN {X 0,Y 282.989,Z 265.705,A -85,B 0,C 180,E1 -18546.591,E2 -18546.591} C_VEL
LIN {X 0,Y 279.353,Z 324.945,A -85,B 0,C 180,E1 -18548.504,E2 -18548.504} C_VEL
LIN {X 0,Y 278.201,Z 337.794,A -85,B 0,C 180,E1 -18549.194,E2 -18549.194} C_VEL
LIN {X 0,Y 276.661,Z 349.845,A -85,B 0,C 180,E1 -18550.106,E2 -18550.106} C_VEL
LIN {X 0,Y 274.73,Z 361.319,A -85,B 0,C 180,E1 -18551.248,E2 -18551.248} C_VEL
LIN {X 0,Y 272.516,Z 372.163,A -85,B 0,C 180,E1 -18552.631,E2 -18552.631} C_VEL
LIN {X 0,Y 270.012,Z 382.561,A -85,B 0,C 180,E1 -18554.295,E2 -18554.295} C_VEL
LIN {X 0,Y 267.679,Z 391.142,A -85,B 0,C 180,E1 -18556.003,E2 -18556.003} C_VEL
LIN {X 0,Y 265.167,Z 399.417,A -85,B 0,C 180,E1 -18558.043,E2 -18558.043} C_VEL
LIN {X 0,Y 262.567,Z 407.175,A -85,B 0,C 180,E1 -18560.475,E2 -18560.475} C_VEL
LIN {X 0,Y 260.567,Z 412.76,A -85,B 0,C 180,E1 -18562.708,E2 -18562.708} C_VEL
LIN {X 0,Y 258.984,Z 417.011,A -85,B 0,C 180,E1 -18564.874,E2 -18564.874} C_VEL
LIN {X 0,Y 257.271,Z 421.087,A -85,B 0,C 180,E1 -18567.671,E2 -18567.671} C_VEL
LIN {X 0,Y 256.352,Z 422.969,A -85,B 0,C 180,E1 -18569.569,E2 -18569.569} C_VEL
LIN {X 0,Y 255.625,Z 424.3,A -85,B 0,C 180,E1 -18571.538,E2 -18571.538} C_VEL
LIN {X 0,Y 254.869,Z 425.053,A -85,B 0,C 180,E1 -18574.184,E2 -18574.184} C_VEL
LIN {X 0,Y 254.459,Z 424.691,A -85,B 0,C 180,E1 -18576.778,E2 -18576.778} C_VEL
LIN {X 0,Y 254.347,Z 423.164,A -85,B 0,C 180,E1 -18579.459,E2 -18579.459} C_VEL
LIN {X 0,Y 254.664,Z 419.82,A -85,B 0,C 180,E1 -18582.63,E2 -18582.63} C_VEL
LIN {X 0,Y 255.087,Z 416.274,A -85,B 0,C 180,E1 -18584.907,E2 -18584.907} C_VEL
LIN {X 0,Y 255.652,Z 411.74,A -85,B 0,C 180,E1 -18587.157,E2 -18587.157} C_VEL
LIN {X 0,Y 256.396,Z 406.11,A -85,B 0,C 180,E1 -18589.386,E2 -18589.386} C_VEL
LIN {X 0,Y 257.412,Z 398.783,A -85,B 0,C 180,E1 -18591.71,E2 -18591.71} C_VEL
LIN {X 0,Y 258.719,Z 390.135,A -85,B 0,C 180,E1 -18593.914,E2 -18593.914} C_VEL
LIN {X 0,Y 259.902,Z 381.471,A -85,B 0,C 180,E1 -18595.721,E2 -18595.721} C_VEL
LIN {X 0,Y 261.236,Z 371.332,A -85,B 0,C 180,E1 -18597.449,E2 -18597.449} C_VEL
LIN {X 0,Y 262.641,Z 359.451,A -85,B 0,C 180,E1 -18599.05,E2 -18599.05} C_VEL
LIN {X 0,Y 263.853,Z 347.583,A -85,B 0,C 180,E1 -18600.301,E2 -18600.301} C_VEL
LIN {X 0,Y 264.892,Z 334.572,A -85,B 0,C 180,E1 -18601.321,E2 -18601.321} C_VEL
LIN {X 0,Y 265.364,Z 323.378,A -85,B 0,C 180,E1 -18601.96,E2 -18601.96} C_VEL
LIN {X 0,Y 266.19,Z 301.997,A -85,B 0,C 180,E1 -18602.695,E2 -18602.695} C_VEL
LIN {X 0,Y 267.902,Z 252.428,A -85,B 0,C 180,E1 -18604.248,E2 -18604.248} C_VEL
LIN {X 0,Y 257.833,Z 227.146,A -85,B 0,C 180,E1 -18605.947,E2 -18605.947} C_VEL
LIN {X 0,Y 256.14,Z 222.58,A -85,B 0,C 180,E1 -18606.288,E2 -18606.288} C_VEL
LIN {X 0,Y 256.159,Z 222.578,A -85,B 0,C 180,E1 -18610.778,E2 -18610.778} C_VEL
LIN {X 0,Y 256.259,Z 222.563,A -85,B 0,C 180,E1 -18614.083,E2 -18614.083} C_VEL
LIN {X 0,Y 256.291,Z 222.562,A -85,B 0,C 180,E1 -18618.934,E2 -18618.934} C_VEL
LIN {X 0,Y 256.471,Z 222.537,A -85,B 0,C 180,E1 -18622.125,E2 -18622.125} C_VEL
LIN {X 0,Y 256.492,Z 222.535,A -85,B 0,C 180,E1 -18626.859,E2 -18626.859} C_VEL
LIN {X 0,Y 256.751,Z 222.501,A -85,B 0,C 180,E1 -18630,E2 -18630} C_VEL
LIN {X 0,Y 256.484,Z 222.534,A -85,B 0,C 180,E1 -18633.142,E2 -18633.142} C_VEL
LIN {X 0,Y 256.497,Z 222.533,A -85,B 0,C 180,E1 -18637.875,E2 -18637.875} C_VEL
LIN {X 0,Y 256.297,Z 222.559,A -85,B 0,C 180,E1 -18642.673,E2 -18642.673} C_VEL
LIN {X 0,Y 256.285,Z 222.562,A -85,B 0,C 180,E1 -18646.303,E2 -18646.303} C_VEL
LIN {X 0,Y 256.155,Z 222.569,A -85,B 0,C 180,E1 -18651.117,E2 -18651.117} C_VEL
LIN {X 0,Y 256.136,Z 222.575,A -85,B 0,C 180,E1 -18655.113,E2 -18655.113} C_VEL
LIN {X 0,Y 256.058,Z 222.59,A -85,B 0,C 180,E1 -18659.607,E2 -18659.607} C_VEL
LIN {X 0,Y 256.068,Z 222.585,A -85,B 0,C 180,E1 -18663.293,E2 -18663.293} C_VEL
LIN {X 0,Y 256.111,Z 222.571,A -85,B 0,C 180,E1 -18667.27,E2 -18667.27} C_VEL
LIN {X 0,Y 256.051,Z 222.582,A -85,B 0,C 180,E1 -18671.205,E2 -18671.205} C_VEL
LIN {X 0,Y 256.041,Z 222.592,A -85,B 0,C 180,E1 -18675.535,E2 -18675.535} C_VEL
LIN {X 0,Y 256.042,Z 222.59,A -85,B 0,C 180,E1 -18678.794,E2 -18678.794} C_VEL
LIN {X 0,Y 256.13,Z 222.576,A -85,B 0,C 180,E1 -18682.867,E2 -18682.867} C_VEL
LIN {X 0,Y 256.068,Z 222.586,A -85,B 0,C 180,E1 -18686.707,E2 -18686.707} C_VEL
LIN {X 0,Y 256.057,Z 222.587,A -85,B 0,C 180,E1 -18690.393,E2 -18690.393} C_VEL
LIN {X 0,Y 256.135,Z 222.577,A -85,B 0,C 180,E1 -18694.889,E2 -18694.889} C_VEL
LIN {X 0,Y 256.151,Z 222.578,A -85,B 0,C 180,E1 -18699.104,E2 -18699.104} C_VEL
LIN {X 0,Y 256.262,Z 222.56,A -85,B 0,C 180,E1 -18704.083,E2 -18704.083} C_VEL
LIN {X 0,Y 256.294,Z 222.546,A -85,B 0,C 180,E1 -18708.933,E2 -18708.933} C_VEL
LIN {X 0,Y 256.472,Z 222.525,A -85,B 0,C 180,E1 -18712.125,E2 -18712.125} C_VEL
LIN {X 0,Y 256.486,Z 222.534,A -85,B 0,C 180,E1 -18716.859,E2 -18716.859} C_VEL
LIN {X 0,Y 256.708,Z 222.51,A -85,B 0,C 180,E1 -18718.431,E2 -18718.431} C_VEL
LIN {X 0,Y 256.703,Z 222.507,A -85,B 0,C 180,E1 -18721.569,E2 -18721.569} C_VEL
LIN {X 0,Y 256.458,Z 222.533,A -85,B 0,C 180,E1 -18726.293,E2 -18726.293} C_VEL
LIN {X 0,Y 256.43,Z 222.534,A -85,B 0,C 180,E1 -18729.465,E2 -18729.465} C_VEL
LIN {X 0,Y 256.287,Z 222.555,A -85,B 0,C 180,E1 -18731.131,E2 -18731.131} C_VEL
LIN {X 0,Y 255.56,Z 222.651,A -85,B 0,C 180,E1 -18732.442,E2 -18732.442} C_VEL
LIN {X 0,Y 252.707,Z 223.008,A -85,B 0,C 180,E1 -18734.578,E2 -18734.578} C_VEL
LIN {X 0,Y 250.294,Z 223.314,A -85,B 0,C 180,E1 -18736.316,E2 -18736.316} C_VEL
LIN {X 0,Y 249.219,Z 223.444,A -85,B 0,C 180,E1 -18737.664,E2 -18737.664} C_VEL
LIN {X 0,Y 249.108,Z 223.454,A -85,B 0,C 180,E1 -18738.12,E2 -18738.12} C_VEL
LIN {X 0,Y 249.08,Z 223.453,A -85,B 0,C 180,E1 -18741.519,E2 -18741.519} C_VEL
LIN {X 0,Y 249.052,Z 223.463,A -85,B 0,C 180,E1 -18745.442,E2 -18745.442} C_VEL
LIN {X 0,Y 249.039,Z 223.462,A -85,B 0,C 180,E1 -18748.973,E2 -18748.973} C_VEL
LIN {X 0,Y 249.03,Z 223.462,A -85,B 0,C 180,E1 -18752.426,E2 -18752.426} C_VEL
LIN {X 0,Y 249.029,Z 223.463,A -85,B 0,C 180,E1 -18756.346,E2 -18756.346} C_VEL
LIN {X 0,Y 248.987,Z 223.47,A -85,B 0,C 180,E1 -18760.482,E2 -18760.482} C_VEL
LIN {X 0,Y 248.964,Z 223.474,A -85,B 0,C 180,E1 -18764.888,E2 -18764.888} C_VEL
LIN {X 0,Y 248.981,Z 223.472,A -85,B 0,C 180,E1 -18767.355,E2 -18767.355} C_VEL
LIN {X 0,Y 249.046,Z 223.463,A -85,B 0,C 180,E1 -18772.2,E2 -18772.2} C_VEL
LIN {X 0,Y 249.11,Z 223.528,A -85,B 0,C 180,E1 -18772.785,E2 -18772.785} C_VEL
LIN {X 0,Y 251.727,Z 235.685,A -85,B 0,C 180,E1 -18776.885,E2 -18776.885} C_VEL
LIN {X 0,Y 254.085,Z 247.216,A -85,B 0,C 180,E1 -18780.596,E2 -18780.596} C_VEL
LIN {X 0,Y 254.125,Z 249.197,A -85,B 0,C 180,E1 -18781.195,E2 -18781.195} C_VEL
LIN {X 0,Y 259.942,Z 305.193,A -85,B 0,C 180,E1 -18783.659,E2 -18783.659} C_VEL
LIN {X 0,Y 258.03,Z 359.254,A -85,B 0,C 180,E1 -18785.457,E2 -18785.457} C_VEL
LIN {X 0,Y 257.056,Z 372.884,A -85,B 0,C 180,E1 -18786.217,E2 -18786.217} C_VEL
LIN {X 0,Y 255.798,Z 384.799,A -85,B 0,C 180,E1 -18787.164,E2 -18787.164} C_VEL
LIN {X 0,Y 254.203,Z 397.295,A -85,B 0,C 180,E1 -18788.51,E2 -18788.51} C_VEL
LIN {X 0,Y 252.663,Z 408.568,A -85,B 0,C 180,E1 -18790.077,E2 -18790.077} C_VEL
LIN {X 0,Y 251.12,Z 418.75,A -85,B 0,C 180,E1 -18791.859,E2 -18791.859} C_VEL
LIN {X 0,Y 249.859,Z 427.134,A -85,B 0,C 180,E1 -18793.663,E2 -18793.663} C_VEL
LIN {X 0,Y 248.743,Z 436.295,A -85,B 0,C 180,E1 -18796.104,E2 -18796.104} C_VEL
LIN {X 0,Y 247.839,Z 443.603,A -85,B 0,C 180,E1 -18798.55,E2 -18798.55} C_VEL
LIN {X 0,Y 247.442,Z 449.395,A -85,B 0,C 180,E1 -18801.012,E2 -18801.012} C_VEL
LIN {X 0,Y 247.389,Z 454.536,A -85,B 0,C 180,E1 -18803.884,E2 -18803.884} C_VEL
LIN {X 0,Y 247.411,Z 456.248,A -85,B 0,C 180,E1 -18805.111,E2 -18805.111} C_VEL
LIN {X 0,Y 247.361,Z 458.112,A -85,B 0,C 180,E1 -18806.742,E2 -18806.742} C_VEL
LIN {X 0,Y 247.535,Z 459.496,A -85,B 0,C 180,E1 -18808.373,E2 -18808.373} C_VEL
LIN {X 0,Y 247.7,Z 460.428,A -85,B 0,C 180,E1 -18810,E2 -18810} C_VEL
LIN {X 0,Y 247.422,Z 460.902,A -85,B 0,C 180,E1 -18811.627,E2 -18811.627} C_VEL
LIN {X 0,Y 247.23,Z 460.965,A -85,B 0,C 180,E1 -18813.259,E2 -18813.259} C_VEL
LIN {X 0,Y 247.04,Z 460.41,A -85,B 0,C 180,E1 -18815.306,E2 -18815.306} C_VEL
LIN {X 0,Y 247.176,Z 458.61,A -85,B 0,C 180,E1 -18818.173,E2 -18818.173} C_VEL
LIN {X 0,Y 247.603,Z 456.041,A -85,B 0,C 180,E1 -18820.631,E2 -18820.631} C_VEL
LIN {X 0,Y 248.43,Z 452.489,A -85,B 0,C 180,E1 -18823.08,E2 -18823.08} C_VEL
LIN {X 0,Y 249.912,Z 447.877,A -85,B 0,C 180,E1 -18825.495,E2 -18825.495} C_VEL
LIN {X 0,Y 252.026,Z 440.936,A -85,B 0,C 180,E1 -18828.33,E2 -18828.33} C_VEL
LIN {X 0,Y 254.26,Z 433.691,A -85,B 0,C 180,E1 -18830.635,E2 -18830.635} C_VEL
LIN {X 0,Y 257.235,Z 424.61,A -85,B 0,C 180,E1 -18832.912,E2 -18832.912} C_VEL
LIN {X 0,Y 260.31,Z 414.394,A -85,B 0,C 180,E1 -18834.951,E2 -18834.951} C_VEL
LIN {X 0,Y 263.517,Z 402.791,A -85,B 0,C 180,E1 -18836.747,E2 -18836.747} C_VEL
LIN {X 0,Y 266.359,Z 391.329,A -85,B 0,C 180,E1 -18838.14,E2 -18838.14} C_VEL
LIN {X 0,Y 269.085,Z 378.373,A -85,B 0,C 180,E1 -18839.321,E2 -18839.321} C_VEL
LIN {X 0,Y 271.357,Z 364.688,A -85,B 0,C 180,E1 -18840.226,E2 -18840.226} C_VEL
LIN {X 0,Y 272.778,Z 350.722,A -85,B 0,C 180,E1 -18840.855,E2 -18840.855} C_VEL
LIN {X 0,Y 275.384,Z 308.222,A -85,B 0,C 180,E1 -18842.241,E2 -18842.241} C_VEL
LIN {X 0,Y 273.973,Z 291.106,A -85,B 0,C 180,E1 -18843.285,E2 -18843.285} C_VEL
LIN {X 0,Y 271.74,Z 273.984,A -85,B 0,C 180,E1 -18844.562,E2 -18844.562} C_VEL
LIN {X 0,Y 270.597,Z 270.567,A -85,B 0,C 180,E1 -18844.976,E2 -18844.976} C_VEL
LIN {X 0,Y 266.179,Z 260.877,A -85,B 0,C 180,E1 -18846.487,E2 -18846.487} C_VEL
LIN {X 0,Y 263.222,Z 255.075,A -85,B 0,C 180,E1 -18847.542,E2 -18847.542} C_VEL
LIN {X 0,Y 260.996,Z 250.944,A -85,B 0,C 180,E1 -18848.356,E2 -18848.356} C_VEL
LIN {X 0,Y 258.152,Z 245.905,A -85,B 0,C 180,E1 -18849.462,E2 -18849.462} C_VEL
LIN {X 0,Y 254.662,Z 240.101,A -85,B 0,C 180,E1 -18850.896,E2 -18850.896} C_VEL
LIN {X 0,Y 252.743,Z 234.121,A -85,B 0,C 180,E1 -18854.04,E2 -18854.04} C_VEL
LIN {X 0,Y 250.635,Z 228.175,A -85,B 0,C 180,E1 -18857.702,E2 -18857.702} C_VEL
LIN {X 0,Y 250.223,Z 226.646,A -85,B 0,C 180,E1 -18858.698,E2 -18858.698} C_VEL
LIN {X 0,Y 249.021,Z 223.467,A -85,B 0,C 180,E1 -18861.23,E2 -18861.23} C_VEL
LIN {X 0,Y 249.043,Z 223.459,A -85,B 0,C 180,E1 -18865.639,E2 -18865.639} C_VEL
LIN {X 0,Y 249.002,Z 223.467,A -85,B 0,C 180,E1 -18869.466,E2 -18869.466} C_VEL
LIN {X 0,Y 249.037,Z 223.457,A -85,B 0,C 180,E1 -18873.158,E2 -18873.158} C_VEL
LIN {X 0,Y 249.056,Z 223.455,A -85,B 0,C 180,E1 -18876.73,E2 -18876.73} C_VEL
LIN {X 0,Y 249.087,Z 223.453,A -85,B 0,C 180,E1 -18880.209,E2 -18880.209} C_VEL
LIN {X 0,Y 249.195,Z 223.441,A -85,B 0,C 180,E1 -18883.619,E2 -18883.619} C_VEL
LIN {X 0,Y 249.243,Z 223.431,A -85,B 0,C 180,E1 -18888.616,E2 -18888.616} C_VEL
LIN {X 0,Y 249.455,Z 223.409,A -85,B 0,C 180,E1 -18891.902,E2 -18891.902} C_VEL
LIN {X 0,Y 249.312,Z 223.431,A -85,B 0,C 180,E1 -18895.351,E2 -18895.351} C_VEL
LIN {X 0,Y 250.082,Z 225.79,A -85,B 0,C 180,E1 -18895.82,E2 -18895.82} C_VEL
LIN {X 0,Y 252.039,Z 228.071,A -85,B 0,C 180,E1 -18896.703,E2 -18896.703} C_VEL
LIN {X 0,Y 253.598,Z 229.104,A -85,B 0,C 180,E1 -18897.325,E2 -18897.325} C_VEL
LIN {X 0,Y 255.596,Z 232.418,A -85,B 0,C 180,E1 -18898.208,E2 -18898.208} C_VEL
LIN {X 0,Y 257.387,Z 234.287,A -85,B 0,C 180,E1 -18898.886,E2 -18898.886} C_VEL
LIN {X 0,Y 259.959,Z 237.985,A -85,B 0,C 180,E1 -18899.88,E2 -18899.88} C_VEL
LIN {X 0,Y 264.262,Z 244.821,A -85,B 0,C 180,E1 -18901.452,E2 -18901.452} C_VEL
LIN {X 0,Y 270.16,Z 253.951,A -85,B 0,C 180,E1 -18903.396,E2 -18903.396} C_VEL
LIN {X 0,Y 276.061,Z 265.038,A -85,B 0,C 180,E1 -18905.206,E2 -18905.206} C_VEL
LIN {X 0,Y 277.563,Z 268.199,A -85,B 0,C 180,E1 -18905.663,E2 -18905.663} C_VEL
LIN {X 0,Y 273.856,Z 326.344,A -85,B 0,C 180,E1 -18907.604,E2 -18907.604} C_VEL
LIN {X 0,Y 272.647,Z 339.064,A -85,B 0,C 180,E1 -18908.314,E2 -18908.314} C_VEL
LIN {X 0,Y 270.894,Z 351.783,A -85,B 0,C 180,E1 -18909.31,E2 -18909.31} C_VEL
LIN {X 0,Y 268.726,Z 363.569,A -85,B 0,C 180,E1 -18910.549,E2 -18910.549} C_VEL
LIN {X 0,Y 266.393,Z 374.066,A -85,B 0,C 180,E1 -18911.955,E2 -18911.955} C_VEL
LIN {X 0,Y 263.716,Z 384.357,A -85,B 0,C 180,E1 -18913.681,E2 -18913.681} C_VEL
LIN {X 0,Y 261.004,Z 393.529,A -85,B 0,C 180,E1 -18915.621,E2 -18915.621} C_VEL
LIN {X 0,Y 258.328,Z 401.736,A -85,B 0,C 180,E1 -18917.788,E2 -18917.788} C_VEL
LIN {X 0,Y 256.067,Z 408.095,A -85,B 0,C 180,E1 -18919.887,E2 -18919.887} C_VEL
LIN {X 0,Y 254.115,Z 413.075,A -85,B 0,C 180,E1 -18921.923,E2 -18921.923} C_VEL
LIN {X 0,Y 251.987,Z 418.359,A -85,B 0,C 180,E1 -18924.731,E2 -18924.731} C_VEL
LIN {X 0,Y 250.227,Z 422.135,A -85,B 0,C 180,E1 -18927.608,E2 -18927.608} C_VEL
LIN {X 0,Y 248.89,Z 424.546,A -85,B 0,C 180,E1 -18930.549,E2 -18930.549} C_VEL
LIN {X 0,Y 248.201,Z 425.398,A -85,B 0,C 180,E1 -18932.547,E2 -18932.547} C_VEL
LIN {X 0,Y 247.689,Z 425.626,A -85,B 0,C 180,E1 -18934.629,E2 -18934.629} C_VEL
LIN {X 0,Y 247.348,Z 424.944,A -85,B 0,C 180,E1 -18937.291,E2 -18937.291} C_VEL
LIN {X 0,Y 247.274,Z 423.233,A -85,B 0,C 180,E1 -18939.88,E2 -18939.88} C_VEL
LIN {X 0,Y 247.636,Z 419.806,A -85,B 0,C 180,E1 -18942.932,E2 -18942.932} C_VEL
LIN {X 0,Y 248.136,Z 415.41,A -85,B 0,C 180,E1 -18945.647,E2 -18945.647} C_VEL
LIN {X 0,Y 248.943,Z 409.409,A -85,B 0,C 180,E1 -18948.429,E2 -18948.429} C_VEL
LIN {X 0,Y 249.994,Z 402.201,A -85,B 0,C 180,E1 -18950.993,E2 -18950.993} C_VEL
LIN {X 0,Y 251.119,Z 394.582,A -85,B 0,C 180,E1 -18953.174,E2 -18953.174} C_VEL
LIN {X 0,Y 252.369,Z 385.985,A -85,B 0,C 180,E1 -18955.188,E2 -18955.188} C_VEL
LIN {X 0,Y 253.83,Z 375.886,A -85,B 0,C 180,E1 -18957.105,E2 -18957.105} C_VEL
LIN {X 0,Y 255.302,Z 363.805,A -85,B 0,C 180,E1 -18958.926,E2 -18958.926} C_VEL
LIN {X 0,Y 256.659,Z 351.547,A -85,B 0,C 180,E1 -18960.357,E2 -18960.357} C_VEL
LIN {X 0,Y 257.8,Z 338.44,A -85,B 0,C 180,E1 -18961.506,E2 -18961.506} C_VEL
LIN {X 0,Y 258.502,Z 325.251,A -85,B 0,C 180,E1 -18962.335,E2 -18962.335} C_VEL
LIN {X 0,Y 259.141,Z 308.948,A -85,B 0,C 180,E1 -18962.951,E2 -18962.951} C_VEL
LIN {X 0,Y 261.192,Z 253.986,A -85,B 0,C 180,E1 -18964.713,E2 -18964.713} C_VEL
LIN {X 0,Y 251.05,Z 228.629,A -85,B 0,C 180,E1 -18966.484,E2 -18966.484} C_VEL
LIN {X 0,Y 249.094,Z 223.625,A -85,B 0,C 180,E1 -18966.844,E2 -18966.844} C_VEL
LIN {X 0,Y 249.087,Z 223.457,A -85,B 0,C 180,E1 -18970.21,E2 -18970.21} C_VEL
LIN {X 0,Y 249.196,Z 223.443,A -85,B 0,C 180,E1 -18973.619,E2 -18973.619} C_VEL
LIN {X 0,Y 249.234,Z 223.441,A -85,B 0,C 180,E1 -18978.616,E2 -18978.616} C_VEL
LIN {X 0,Y 249.42,Z 223.415,A -85,B 0,C 180,E1 -18981.901,E2 -18981.901} C_VEL
LIN {X 0,Y 249.283,Z 223.432,A -85,B 0,C 180,E1 -18985.149,E2 -18985.149} C_VEL
LIN {X 0,Y 249.674,Z 223.385,A -85,B 0,C 180,E1 -18988.387,E2 -18988.387} C_VEL
LIN {X 0,Y 249.671,Z 223.382,A -85,B 0,C 180,E1 -18991.613,E2 -18991.613} C_VEL
LIN {X 0,Y 249.436,Z 223.415,A -85,B 0,C 180,E1 -18996.472,E2 -18996.472} C_VEL
LIN {X 0,Y 249.345,Z 223.424,A -85,B 0,C 180,E1 -18999.737,E2 -18999.737} C_VEL
LIN {X 0,Y 249.208,Z 223.441,A -85,B 0,C 180,E1 -19004.704,E2 -19004.704} C_VEL
LIN {X 0,Y 249.14,Z 223.451,A -85,B 0,C 180,E1 -19008.078,E2 -19008.078} C_VEL
LIN {X 0,Y 249.085,Z 223.45,A -85,B 0,C 180,E1 -19011.519,E2 -19011.519} C_VEL
LIN {X 0,Y 249.088,Z 223.454,A -85,B 0,C 180,E1 -19015.461,E2 -19015.461} C_VEL
LIN {X 0,Y 249.041,Z 223.462,A -85,B 0,C 180,E1 -19018.975,E2 -19018.975} C_VEL
LIN {X 0,Y 249.029,Z 223.46,A -85,B 0,C 180,E1 -19022.427,E2 -19022.427} C_VEL
LIN {X 0,Y 249.028,Z 223.451,A -85,B 0,C 180,E1 -19026.346,E2 -19026.346} C_VEL
LIN {X 0,Y 248.991,Z 223.459,A -85,B 0,C 180,E1 -19030.482,E2 -19030.482} C_VEL
LIN {X 0,Y 249,Z 223.462,A -85,B 0,C 180,E1 -19032.79,E2 -19032.79} C_VEL
